LIN {X 0,Y 574.061,Z 827.419,A -85,B 0,C 180,E1 26876.471,E2 26876.471} C_VEL
LIN {X 0,Y 574.2,Z 764.795,A -85,B 0,C 180,E1 26875.555,E2 26875.555} C_VEL
LIN {X 0,Y 573.221,Z 758.441,A -85,B 0,C 180,E1 26875.376,E2 26875.376} C_VEL
LIN {X 0,Y 574.18,Z 705.798,A -85,B 0,C 180,E1 26872.197,E2 26872.197} C_VEL
LIN {X 0,Y 574.377,Z 695.779,A -85,B 0,C 180,E1 26871.578,E2 26871.578} C_VEL
LIN {X 0,Y 575.933,Z 695.849,A -85,B 0,C 180,E1 26871.383,E2 26871.383} C_VEL
LIN {X 0,Y 578.516,Z 693.344,A -85,B 0,C 180,E1 26871.064,E2 26871.064} C_VEL
LIN {X 0,Y 581.773,Z 687.657,A -85,B 0,C 180,E1 26870.669,E2 26870.669} C_VEL
LIN {X 0,Y 581.964,Z 745.865,A -85,B 0,C 180,E1 26870.646,E2 26870.646} C_VEL
LIN {X 0,Y 583.12,Z 759.023,A -85,B 0,C 180,E1 26870.508,E2 26870.508} C_VEL
LIN {X 0,Y 585.252,Z 769.853,A -85,B 0,C 180,E1 26870.255,E2 26870.255} C_VEL
LIN {X 0,Y 588.38,Z 779.136,A -85,B 0,C 180,E1 26869.89,E2 26869.89} C_VEL
LIN {X 0,Y 592.368,Z 786.864,A -85,B 0,C 180,E1 26869.429,E2 26869.429} C_VEL
LIN {X 0,Y 594.678,Z 791.282,A -85,B 0,C 180,E1 26868.994,E2 26868.994} C_VEL
LIN {X 0,Y 595.801,Z 794.66,A -85,B 0,C 180,E1 26868.457,E2 26868.457} C_VEL
LIN {X 0,Y 595.651,Z 796.735,A -85,B 0,C 180,E1 26867.897,E2 26867.897} C_VEL
LIN {X 0,Y 594.355,Z 797.607,A -85,B 0,C 180,E1 26867.317,E2 26867.317} C_VEL
LIN {X 0,Y 591.913,Z 797.089,A -85,B 0,C 180,E1 26866.722,E2 26866.722} C_VEL
LIN {X 0,Y 588.782,Z 795.144,A -85,B 0,C 180,E1 26866.197,E2 26866.197} C_VEL
LIN {X 0,Y 584.208,Z 790.552,A -85,B 0,C 180,E1 26865.535,E2 26865.535} C_VEL
LIN {X 0,Y 580.364,Z 783.96,A -85,B 0,C 180,E1 26864.799,E2 26864.799} C_VEL
LIN {X 0,Y 577.598,Z 774.842,A -85,B 0,C 180,E1 26863.96,E2 26863.96} C_VEL
LIN {X 0,Y 576.214,Z 763.514,A -85,B 0,C 180,E1 26863.07,E2 26863.07} C_VEL
LIN {X 0,Y 576.201,Z 743.269,A -85,B 0,C 180,E1 26861.695,E2 26861.695} C_VEL
LIN {X 0,Y 577.123,Z 706.105,A -85,B 0,C 180,E1 26859.16,E2 26859.16} C_VEL
LIN {X 0,Y 577.781,Z 682.335,A -85,B 0,C 180,E1 26857.465,E2 26857.465} C_VEL
LIN {X 0,Y 572.74,Z 672.999,A -85,B 0,C 180,E1 26856.161,E2 26856.161} C_VEL
LIN {X 0,Y 570.173,Z 668.299,A -85,B 0,C 180,E1 26855.481,E2 26855.481} C_VEL
LIN {X 0,Y 568.395,Z 664.903,A -85,B 0,C 180,E1 26854.992,E2 26854.992} C_VEL
LIN {X 0,Y 568.214,Z 663.961,A -85,B 0,C 180,E1 26854.882,E2 26854.882} C_VEL
LIN {X 0,Y 568.211,Z 663.959,A -85,B 0,C 180,E1 26851.607,E2 26851.607} C_VEL
LIN {X 0,Y 568.205,Z 663.957,A -85,B 0,C 180,E1 26848.252,E2 26848.252} C_VEL
LIN {X 0,Y 568.203,Z 663.955,A -85,B 0,C 180,E1 26844.981,E2 26844.981} C_VEL
LIN {X 0,Y 568.209,Z 663.955,A -85,B 0,C 180,E1 26841.686,E2 26841.686} C_VEL
LIN {X 0,Y 568.205,Z 663.957,A -85,B 0,C 180,E1 26838.466,E2 26838.466} C_VEL
LIN {X 0,Y 568.22,Z 663.957,A -85,B 0,C 180,E1 26835.2,E2 26835.2} C_VEL
LIN {X 0,Y 568.219,Z 663.959,A -85,B 0,C 180,E1 26831.881,E2 26831.881} C_VEL
LIN {X 0,Y 568.204,Z 663.958,A -85,B 0,C 180,E1 26828.602,E2 26828.602} C_VEL
LIN {X 0,Y 568.207,Z 663.956,A -85,B 0,C 180,E1 26825.351,E2 26825.351} C_VEL
LIN {X 0,Y 568.2,Z 663.956,A -85,B 0,C 180,E1 26822.118,E2 26822.118} C_VEL
LIN {X 0,Y 568.201,Z 663.956,A -85,B 0,C 180,E1 26818.891,E2 26818.891} C_VEL
LIN {X 0,Y 568.2,Z 663.956,A -85,B 0,C 180,E1 26815.66,E2 26815.66} C_VEL
LIN {X 0,Y 568.2,Z 663.957,A -85,B 0,C 180,E1 26812.416,E2 26812.416} C_VEL
LIN {X 0,Y 568.209,Z 663.957,A -85,B 0,C 180,E1 26809.147,E2 26809.147} C_VEL
LIN {X 0,Y 568.212,Z 663.958,A -85,B 0,C 180,E1 26805.842,E2 26805.842} C_VEL
LIN {X 0,Y 568.217,Z 663.957,A -85,B 0,C 180,E1 26802.488,E2 26802.488} C_VEL
LIN {X 0,Y 568.211,Z 663.955,A -85,B 0,C 180,E1 26799.815,E2 26799.815} C_VEL
LIN {X 0,Y 567.229,Z 664.083,A -85,B 0,C 180,E1 26799.039,E2 26799.039} C_VEL
LIN {X 0,Y 560.723,Z 664.89,A -85,B 0,C 180,E1 26796.802,E2 26796.802} C_VEL
LIN {X 0,Y 560.27,Z 664.947,A -85,B 0,C 180,E1 26796.29,E2 26796.29} C_VEL
LIN {X 0,Y 560.272,Z 664.94,A -85,B 0,C 180,E1 26793.045,E2 26793.045} C_VEL
LIN {X 0,Y 560.263,Z 664.941,A -85,B 0,C 180,E1 26789.74,E2 26789.74} C_VEL
LIN {X 0,Y 560.264,Z 664.943,A -85,B 0,C 180,E1 26786.45,E2 26786.45} C_VEL
LIN {X 0,Y 560.265,Z 664.941,A -85,B 0,C 180,E1 26783.156,E2 26783.156} C_VEL
LIN {X 0,Y 560.267,Z 664.943,A -85,B 0,C 180,E1 26779.891,E2 26779.891} C_VEL
LIN {X 0,Y 560.276,Z 664.948,A -85,B 0,C 180,E1 26776.578,E2 26776.578} C_VEL
LIN {X 0,Y 560.285,Z 664.95,A -85,B 0,C 180,E1 26773.256,E2 26773.256} C_VEL
LIN {X 0,Y 560.279,Z 664.95,A -85,B 0,C 180,E1 26769.84,E2 26769.84} C_VEL
LIN {X 0,Y 560.292,Z 665.024,A -85,B 0,C 180,E1 26767.165,E2 26767.165} C_VEL
LIN {X 0,Y 566.144,Z 680.018,A -85,B 0,C 180,E1 26765.71,E2 26765.71} C_VEL
LIN {X 0,Y 565.24,Z 725.275,A -85,B 0,C 180,E1 26762.648,E2 26762.648} C_VEL
LIN {X 0,Y 564.523,Z 766.047,A -85,B 0,C 180,E1 26759.972,E2 26759.972} C_VEL
LIN {X 0,Y 565.697,Z 774.516,A -85,B 0,C 180,E1 26759.782,E2 26759.782} C_VEL
LIN {X 0,Y 564.529,Z 1010.135,A -85,B 0,C 180,E1 26756.517,E2 26756.517} C_VEL
LIN {X 0,Y 564.318,Z 1034.29,A -85,B 0,C 180,E1 26756.118,E2 26756.118} C_VEL
LIN {X 0,Y 563.978,Z 1055.272,A -85,B 0,C 180,E1 26755.57,E2 26755.57} C_VEL
LIN {X 0,Y 563.594,Z 1074.97,A -85,B 0,C 180,E1 26754.863,E2 26754.863} C_VEL
LIN {X 0,Y 563.134,Z 1093.888,A -85,B 0,C 180,E1 26753.991,E2 26753.991} C_VEL
LIN {X 0,Y 562.646,Z 1111.983,A -85,B 0,C 180,E1 26752.964,E2 26752.964} C_VEL
LIN {X 0,Y 562.137,Z 1130.277,A -85,B 0,C 180,E1 26751.713,E2 26751.713} C_VEL
LIN {X 0,Y 561.654,Z 1147.441,A -85,B 0,C 180,E1 26750.312,E2 26750.312} C_VEL
LIN {X 0,Y 561.203,Z 1163.492,A -85,B 0,C 180,E1 26748.763,E2 26748.763} C_VEL
LIN {X 0,Y 560.824,Z 1178.065,A -85,B 0,C 180,E1 26747.107,E2 26747.107} C_VEL
LIN {X 0,Y 560.51,Z 1191.489,A -85,B 0,C 180,E1 26745.307,E2 26745.307} C_VEL
LIN {X 0,Y 560.275,Z 1203.372,A -85,B 0,C 180,E1 26743.414,E2 26743.414} C_VEL
LIN {X 0,Y 560.11,Z 1213.696,A -85,B 0,C 180,E1 26741.428,E2 26741.428} C_VEL
LIN {X 0,Y 560.004,Z 1222.013,A -85,B 0,C 180,E1 26739.454,E2 26739.454} C_VEL
LIN {X 0,Y 559.938,Z 1228.879,A -85,B 0,C 180,E1 26737.386,E2 26737.386} C_VEL
LIN {X 0,Y 559.914,Z 1234.17,A -85,B 0,C 180,E1 26735.225,E2 26735.225} C_VEL
LIN {X 0,Y 559.913,Z 1237.506,A -85,B 0,C 180,E1 26733.173,E2 26733.173} C_VEL
LIN {X 0,Y 559.912,Z 1239.241,A -85,B 0,C 180,E1 26731.125,E2 26731.125} C_VEL
LIN {X 0,Y 559.914,Z 1239.294,A -85,B 0,C 180,E1 26728.976,E2 26728.976} C_VEL
LIN {X 0,Y 559.914,Z 1237.717,A -85,B 0,C 180,E1 26726.929,E2 26726.929} C_VEL
LIN {X 0,Y 559.914,Z 1234.347,A -85,B 0,C 180,E1 26724.774,E2 26724.774} C_VEL
LIN {X 0,Y 559.934,Z 1229.439,A -85,B 0,C 180,E1 26722.716,E2 26722.716} C_VEL
LIN {X 0,Y 559.991,Z 1222.758,A -85,B 0,C 180,E1 26720.649,E2 26720.649} C_VEL
LIN {X 0,Y 560.099,Z 1214.577,A -85,B 0,C 180,E1 26718.675,E2 26718.675} C_VEL
LIN {X 0,Y 560.243,Z 1205.016,A -85,B 0,C 180,E1 26716.794,E2 26716.794} C_VEL
LIN {X 0,Y 560.463,Z 1193.494,A -85,B 0,C 180,E1 26714.902,E2 26714.902} C_VEL
LIN {X 0,Y 560.762,Z 1180.465,A -85,B 0,C 180,E1 26713.104,E2 26713.104} C_VEL
LIN {X 0,Y 561.151,Z 1165.383,A -85,B 0,C 180,E1 26711.347,E2 26711.347} C_VEL
LIN {X 0,Y 561.596,Z 1149.282,A -85,B 0,C 180,E1 26709.763,E2 26709.763} C_VEL
LIN {X 0,Y 562.058,Z 1132.894,A -85,B 0,C 180,E1 26708.393,E2 26708.393} C_VEL
LIN {X 0,Y 562.578,Z 1115.255,A -85,B 0,C 180,E1 26707.149,E2 26707.149} C_VEL
LIN {X 0,Y 563.08,Z 1096.267,A -85,B 0,C 180,E1 26706.042,E2 26706.042} C_VEL
LIN {X 0,Y 563.532,Z 1076.995,A -85,B 0,C 180,E1 26705.133,E2 26705.133} C_VEL
LIN {X 0,Y 563.952,Z 1056.45,A -85,B 0,C 180,E1 26704.378,E2 26704.378} C_VEL
LIN {X 0,Y 564.303,Z 1035.559,A -85,B 0,C 180,E1 26703.82,E2 26703.82} C_VEL
LIN {X 0,Y 564.518,Z 1012.48,A -85,B 0,C 180,E1 26703.425,E2 26703.425} C_VEL
LIN {X 0,Y 565.69,Z 776.957,A -85,B 0,C 180,E1 26700.162,E2 26700.162} C_VEL
LIN {X 0,Y 563.542,Z 767.47,A -85,B 0,C 180,E1 26699.888,E2 26699.888} C_VEL
LIN {X 0,Y 564.325,Z 733.661,A -85,B 0,C 180,E1 26696.684,E2 26696.684} C_VEL
LIN {X 0,Y 565.011,Z 702.166,A -85,B 0,C 180,E1 26693.628,E2 26693.628} C_VEL
LIN {X 0,Y 565.36,Z 679.55,A -85,B 0,C 180,E1 26691.416,E2 26691.416} C_VEL
LIN {X 0,Y 560.271,Z 664.95,A -85,B 0,C 180,E1 26689.556,E2 26689.556} C_VEL
LIN {X 0,Y 560.272,Z 664.947,A -85,B 0,C 180,E1 26686.178,E2 26686.178} C_VEL
LIN {X 0,Y 560.267,Z 664.94,A -85,B 0,C 180,E1 26682.821,E2 26682.821} C_VEL
LIN {X 0,Y 560.281,Z 664.944,A -85,B 0,C 180,E1 26679.401,E2 26679.401} C_VEL
LIN {X 0,Y 560.283,Z 664.949,A -85,B 0,C 180,E1 26675.953,E2 26675.953} C_VEL
LIN {X 0,Y 560.289,Z 665.066,A -85,B 0,C 180,E1 26674.08,E2 26674.08} C_VEL
LIN {X 0,Y 565.192,Z 678.885,A -85,B 0,C 180,E1 26672.474,E2 26672.474} C_VEL
LIN {X 0,Y 563.991,Z 718.046,A -85,B 0,C 180,E1 26669.12,E2 26669.12} C_VEL
LIN {X 0,Y 563.138,Z 756.776,A -85,B 0,C 180,E1 26665.955,E2 26665.955} C_VEL
LIN {X 0,Y 562.433,Z 797.021,A -85,B 0,C 180,E1 26662.762,E2 26662.762} C_VEL
LIN {X 0,Y 561.797,Z 839.094,A -85,B 0,C 180,E1 26659.494,E2 26659.494} C_VEL
LIN {X 0,Y 561.794,Z 845.338,A -85,B 0,C 180,E1 26659.043,E2 26659.043} C_VEL
LIN {X 0,Y 562.522,Z 852.682,A -85,B 0,C 180,E1 26658.919,E2 26658.919} C_VEL
LIN {X 0,Y 561.965,Z 1014.791,A -85,B 0,C 180,E1 26656.766,E2 26656.766} C_VEL
LIN {X 0,Y 561.803,Z 1032.643,A -85,B 0,C 180,E1 26656.339,E2 26656.339} C_VEL
LIN {X 0,Y 561.572,Z 1048.909,A -85,B 0,C 180,E1 26655.755,E2 26655.755} C_VEL
LIN {X 0,Y 561.319,Z 1064.386,A -85,B 0,C 180,E1 26655.021,E2 26655.021} C_VEL
LIN {X 0,Y 561.035,Z 1079.974,A -85,B 0,C 180,E1 26654.08,E2 26654.08} C_VEL
LIN {X 0,Y 560.761,Z 1094.334,A -85,B 0,C 180,E1 26652.983,E2 26652.983} C_VEL
LIN {X 0,Y 560.523,Z 1107.266,A -85,B 0,C 180,E1 26651.786,E2 26651.786} C_VEL
LIN {X 0,Y 560.306,Z 1119.603,A -85,B 0,C 180,E1 26650.384,E2 26650.384} C_VEL
LIN {X 0,Y 560.145,Z 1129.955,A -85,B 0,C 180,E1 26648.934,E2 26648.934} C_VEL
LIN {X 0,Y 560.038,Z 1138.965,A -85,B 0,C 180,E1 26647.386,E2 26647.386} C_VEL
LIN {X 0,Y 559.961,Z 1146.839,A -85,B 0,C 180,E1 26645.636,E2 26645.636} C_VEL
LIN {X 0,Y 559.93,Z 1152.371,A -85,B 0,C 180,E1 26643.994,E2 26643.994} C_VEL
LIN {X 0,Y 559.915,Z 1156.495,A -85,B 0,C 180,E1 26642.252,E2 26642.252} C_VEL
LIN {X 0,Y 559.916,Z 1158.797,A -85,B 0,C 180,E1 26640.512,E2 26640.512} C_VEL
LIN {X 0,Y 559.913,Z 1159.457,A -85,B 0,C 180,E1 26638.772,E2 26638.772} C_VEL
LIN {X 0,Y 559.913,Z 1158.352,A -85,B 0,C 180,E1 26636.929,E2 26636.929} C_VEL
LIN {X 0,Y 559.921,Z 1155.476,A -85,B 0,C 180,E1 26635.158,E2 26635.158} C_VEL
LIN {X 0,Y 559.934,Z 1151.257,A -85,B 0,C 180,E1 26633.541,E2 26633.541} C_VEL
LIN {X 0,Y 559.975,Z 1145.334,A -85,B 0,C 180,E1 26631.891,E2 26631.891} C_VEL
LIN {X 0,Y 560.047,Z 1137.357,A -85,B 0,C 180,E1 26630.229,E2 26630.229} C_VEL
LIN {X 0,Y 560.163,Z 1128.687,A -85,B 0,C 180,E1 26628.781,E2 26628.781} C_VEL
LIN {X 0,Y 560.348,Z 1117.102,A -85,B 0,C 180,E1 26627.217,E2 26627.217} C_VEL
LIN {X 0,Y 560.556,Z 1105.086,A -85,B 0,C 180,E1 26625.909,E2 26625.909} C_VEL
LIN {X 0,Y 560.804,Z 1092.283,A -85,B 0,C 180,E1 26624.753,E2 26624.753} C_VEL
LIN {X 0,Y 561.11,Z 1076.384,A -85,B 0,C 180,E1 26623.595,E2 26623.595} C_VEL
LIN {X 0,Y 561.365,Z 1061.702,A -85,B 0,C 180,E1 26622.749,E2 26622.749} C_VEL
LIN {X 0,Y 561.612,Z 1046.666,A -85,B 0,C 180,E1 26622.062,E2 26622.062} C_VEL
LIN {X 0,Y 561.851,Z 1028.62,A -85,B 0,C 180,E1 26621.459,E2 26621.459} C_VEL
LIN {X 0,Y 561.993,Z 1012.392,A -85,B 0,C 180,E1 26621.104,E2 26621.104} C_VEL
LIN {X 0,Y 562.344,Z 849.073,A -85,B 0,C 180,E1 26618.937,E2 26618.937} C_VEL
LIN {X 0,Y 561.734,Z 844.641,A -85,B 0,C 180,E1 26618.843,E2 26618.843} C_VEL
LIN {X 0,Y 562.377,Z 801.196,A -85,B 0,C 180,E1 26615.476,E2 26615.476} C_VEL
LIN {X 0,Y 563.114,Z 758.703,A -85,B 0,C 180,E1 26612.11,E2 26612.11} C_VEL
LIN {X 0,Y 563.618,Z 737.518,A -85,B 0,C 180,E1 26610.373,E2 26610.373} C_VEL
LIN {X 0,Y 566.841,Z 712.359,A -85,B 0,C 180,E1 26607.812,E2 26607.812} C_VEL
LIN {X 0,Y 571.277,Z 691.502,A -85,B 0,C 180,E1 26605.523,E2 26605.523} C_VEL
LIN {X 0,Y 572.681,Z 686.32,A -85,B 0,C 180,E1 26604.881,E2 26604.881} C_VEL
LIN {X 0,Y 571.086,Z 683.566,A -85,B 0,C 180,E1 26603.343,E2 26603.343} C_VEL
LIN {X 0,Y 571.107,Z 682.763,A -85,B 0,C 180,E1 26602.338,E2 26602.338} C_VEL
LIN {X 0,Y 571.316,Z 684.023,A -85,B 0,C 180,E1 26601.526,E2 26601.526} C_VEL
LIN {X 0,Y 571.112,Z 684.711,A -85,B 0,C 180,E1 26601.425,E2 26601.425} C_VEL
LIN {X 0,Y 567.688,Z 695.309,A -85,B 0,C 180,E1 26600.563,E2 26600.563} C_VEL
LIN {X 0,Y 565.443,Z 708.541,A -85,B 0,C 180,E1 26599.652,E2 26599.652} C_VEL
LIN {X 0,Y 563.893,Z 729.692,A -85,B 0,C 180,E1 26598.398,E2 26598.398} C_VEL
LIN {X 0,Y 564.008,Z 751.659,A -85,B 0,C 180,E1 26597.175,E2 26597.175} C_VEL
LIN {X 0,Y 565.908,Z 767.995,A -85,B 0,C 180,E1 26596.235,E2 26596.235} C_VEL
LIN {X 0,Y 569.138,Z 779.936,A -85,B 0,C 180,E1 26595.496,E2 26595.496} C_VEL
LIN {X 0,Y 573.479,Z 789.298,A -85,B 0,C 180,E1 26594.869,E2 26594.869} C_VEL
LIN {X 0,Y 578.552,Z 796.38,A -85,B 0,C 180,E1 26594.318,E2 26594.318} C_VEL
LIN {X 0,Y 582.873,Z 800.653,A -85,B 0,C 180,E1 26593.907,E2 26593.907} C_VEL
LIN {X 0,Y 586.666,Z 803.361,A -85,B 0,C 180,E1 26593.445,E2 26593.445} C_VEL
LIN {X 0,Y 589.834,Z 804.737,A -85,B 0,C 180,E1 26592.92,E2 26592.92} C_VEL
LIN {X 0,Y 592.243,Z 804.795,A -85,B 0,C 180,E1 26592.315,E2 26592.315} C_VEL
LIN {X 0,Y 593.403,Z 803.535,A -85,B 0,C 180,E1 26591.718,E2 26591.718} C_VEL
LIN {X 0,Y 593.289,Z 801.151,A -85,B 0,C 180,E1 26591.149,E2 26591.149} C_VEL
LIN {X 0,Y 591.814,Z 797.58,A -85,B 0,C 180,E1 26590.617,E2 26590.617} C_VEL
LIN {X 0,Y 589.03,Z 792.986,A -85,B 0,C 180,E1 26590.185,E2 26590.185} C_VEL
LIN {X 0,Y 584.618,Z 784.743,A -85,B 0,C 180,E1 26589.67,E2 26589.67} C_VEL
LIN {X 0,Y 581.163,Z 775.111,A -85,B 0,C 180,E1 26589.257,E2 26589.257} C_VEL
LIN {X 0,Y 578.719,Z 764.246,A -85,B 0,C 180,E1 26588.96,E2 26588.96} C_VEL
LIN {X 0,Y 577.209,Z 751.284,A -85,B 0,C 180,E1 26588.775,E2 26588.775} C_VEL
LIN {X 0,Y 576.744,Z 738.293,A -85,B 0,C 180,E1 26588.717,E2 26588.717} C_VEL
LIN {X 0,Y 576.681,Z 705.582,A -85,B 0,C 180,E1 26588.709,E2 26588.709} C_VEL
LIN {X 0,Y 572.755,Z 714.129,A -85,B 0,C 180,E1 26588.217,E2 26588.217} C_VEL
LIN {X 0,Y 569.752,Z 718.329,A -85,B 0,C 180,E1 26587.832,E2 26587.832} C_VEL
LIN {X 0,Y 568.223,Z 719.281,A -85,B 0,C 180,E1 26587.632,E2 26587.632} C_VEL
LIN {X 0,Y 567.239,Z 719.066,A -85,B 0,C 180,E1 26587.502,E2 26587.502} C_VEL
LIN {X 0,Y 566.472,Z 759.406,A -85,B 0,C 180,E1 26585.065,E2 26585.065} C_VEL
LIN {X 0,Y 567.771,Z 768.747,A -85,B 0,C 180,E1 26584.832,E2 26584.832} C_VEL
LIN {X 0,Y 566.351,Z 1004.078,A -85,B 0,C 180,E1 26581.438,E2 26581.438} C_VEL
LIN {X 0,Y 565.933,Z 1066.266,A -85,B 0,C 180,E1 26580.527,E2 26580.527} C_VEL
LIN {X 0,Y 565.555,Z 1088.579,A -85,B 0,C 180,E1 26580.002,E2 26580.002} C_VEL
LIN {X 0,Y 565.047,Z 1110.998,A -85,B 0,C 180,E1 26579.265,E2 26579.265} C_VEL
LIN {X 0,Y 564.539,Z 1131.562,A -85,B 0,C 180,E1 26578.395,E2 26578.395} C_VEL
LIN {X 0,Y 563.916,Z 1151.757,A -85,B 0,C 180,E1 26577.337,E2 26577.337} C_VEL
LIN {X 0,Y 563.287,Z 1171.672,A -85,B 0,C 180,E1 26576.082,E2 26576.082} C_VEL
LIN {X 0,Y 562.667,Z 1190.469,A -85,B 0,C 180,E1 26574.683,E2 26574.683} C_VEL
LIN {X 0,Y 562.059,Z 1208.4,A -85,B 0,C 180,E1 26573.118,E2 26573.118} C_VEL
LIN {X 0,Y 561.559,Z 1224.188,A -85,B 0,C 180,E1 26571.518,E2 26571.518} C_VEL
LIN {X 0,Y 561.086,Z 1239.886,A -85,B 0,C 180,E1 26569.682,E2 26569.682} C_VEL
LIN {X 0,Y 560.71,Z 1254.044,A -85,B 0,C 180,E1 26567.754,E2 26567.754} C_VEL
LIN {X 0,Y 560.408,Z 1266.743,A -85,B 0,C 180,E1 26565.736,E2 26565.736} C_VEL
LIN {X 0,Y 560.192,Z 1277.859,A -85,B 0,C 180,E1 26563.627,E2 26563.627} C_VEL
LIN {X 0,Y 560.053,Z 1287.491,A -85,B 0,C 180,E1 26561.43,E2 26561.43} C_VEL
LIN {X 0,Y 559.975,Z 1295.228,A -85,B 0,C 180,E1 26559.248,E2 26559.248} C_VEL
LIN {X 0,Y 559.928,Z 1300.904,A -85,B 0,C 180,E1 26557.181,E2 26557.181} C_VEL
LIN {X 0,Y 559.906,Z 1305.479,A -85,B 0,C 180,E1 26554.918,E2 26554.918} C_VEL
LIN {X 0,Y 559.9,Z 1308.314,A -85,B 0,C 180,E1 26552.662,E2 26552.662} C_VEL
LIN {X 0,Y 559.894,Z 1309.395,A -85,B 0,C 180,E1 26550.512,E2 26550.512} C_VEL
LIN {X 0,Y 559.899,Z 1308.894,A -85,B 0,C 180,E1 26548.158,E2 26548.158} C_VEL
LIN {X 0,Y 559.9,Z 1306.853,A -85,B 0,C 180,E1 26546.007,E2 26546.007} C_VEL
LIN {X 0,Y 559.908,Z 1303.407,A -85,B 0,C 180,E1 26543.953,E2 26543.953} C_VEL
LIN {X 0,Y 559.942,Z 1297.983,A -85,B 0,C 180,E1 26541.684,E2 26541.684} C_VEL
LIN {X 0,Y 560.003,Z 1291.416,A -85,B 0,C 180,E1 26539.612,E2 26539.612} C_VEL
LIN {X 0,Y 560.111,Z 1282.696,A -85,B 0,C 180,E1 26537.422,E2 26537.422} C_VEL
LIN {X 0,Y 560.286,Z 1272.365,A -85,B 0,C 180,E1 26535.289,E2 26535.289} C_VEL
LIN {X 0,Y 560.529,Z 1261.619,A -85,B 0,C 180,E1 26533.418,E2 26533.418} C_VEL
LIN {X 0,Y 560.865,Z 1248.037,A -85,B 0,C 180,E1 26531.392,E2 26531.392} C_VEL
LIN {X 0,Y 561.288,Z 1232.807,A -85,B 0,C 180,E1 26529.456,E2 26529.456} C_VEL
LIN {X 0,Y 561.785,Z 1217.032,A -85,B 0,C 180,E1 26527.723,E2 26527.723} C_VEL
LIN {X 0,Y 562.372,Z 1199.159,A -85,B 0,C 180,E1 26526.043,E2 26526.043} C_VEL
LIN {X 0,Y 562.97,Z 1181.221,A -85,B 0,C 180,E1 26524.602,E2 26524.602} C_VEL
LIN {X 0,Y 563.597,Z 1161.906,A -85,B 0,C 180,E1 26523.275,E2 26523.275} C_VEL
LIN {X 0,Y 564.221,Z 1141.648,A -85,B 0,C 180,E1 26522.107,E2 26522.107} C_VEL
LIN {X 0,Y 564.832,Z 1120.938,A -85,B 0,C 180,E1 26521.131,E2 26521.131} C_VEL
LIN {X 0,Y 565.313,Z 1099.125,A -85,B 0,C 180,E1 26520.319,E2 26520.319} C_VEL
LIN {X 0,Y 565.78,Z 1076.989,A -85,B 0,C 180,E1 26519.7,E2 26519.7} C_VEL
LIN {X 0,Y 566.051,Z 1054.545,A -85,B 0,C 180,E1 26519.277,E2 26519.277} C_VEL
LIN {X 0,Y 567.388,Z 827.927,A -85,B 0,C 180,E1 26516.031,E2 26516.031} C_VEL
LIN {X 0,Y 567.58,Z 766.128,A -85,B 0,C 180,E1 26515.115,E2 26515.115} C_VEL
LIN {X 0,Y 566.384,Z 758.441,A -85,B 0,C 180,E1 26514.897,E2 26514.897} C_VEL
LIN {X 0,Y 567.303,Z 719.089,A -85,B 0,C 180,E1 26512.488,E2 26512.488} C_VEL
LIN {X 0,Y 568.829,Z 719.046,A -85,B 0,C 180,E1 26512.289,E2 26512.289} C_VEL
LIN {X 0,Y 571.437,Z 716.257,A -85,B 0,C 180,E1 26511.951,E2 26511.951} C_VEL
LIN {X 0,Y 575.154,Z 709.281,A -85,B 0,C 180,E1 26511.481,E2 26511.481} C_VEL
LIN {X 0,Y 576.739,Z 705.432,A -85,B 0,C 180,E1 26511.283,E2 26511.283} C_VEL
LIN {X 0,Y 576.939,Z 746.497,A -85,B 0,C 180,E1 26511.259,E2 26511.259} C_VEL
LIN {X 0,Y 578.105,Z 760.159,A -85,B 0,C 180,E1 26511.115,E2 26511.115} C_VEL
LIN {X 0,Y 580.288,Z 771.863,A -85,B 0,C 180,E1 26510.848,E2 26510.848} C_VEL
LIN {X 0,Y 583.457,Z 781.953,A -85,B 0,C 180,E1 26510.468,E2 26510.468} C_VEL
LIN {X 0,Y 587.575,Z 790.606,A -85,B 0,C 180,E1 26509.984,E2 26509.984} C_VEL
LIN {X 0,Y 591.165,Z 796.381,A -85,B 0,C 180,E1 26509.515,E2 26509.515} C_VEL
LIN {X 0,Y 593,Z 800.231,A -85,B 0,C 180,E1 26509.013,E2 26509.013} C_VEL
LIN {X 0,Y 593.488,Z 803.086,A -85,B 0,C 180,E1 26508.418,E2 26508.418} C_VEL
LIN {X 0,Y 592.548,Z 804.664,A -85,B 0,C 180,E1 26507.796,E2 26507.796} C_VEL
LIN {X 0,Y 590.294,Z 804.841,A -85,B 0,C 180,E1 26507.174,E2 26507.174} C_VEL
LIN {X 0,Y 587.239,Z 803.679,A -85,B 0,C 180,E1 26506.637,E2 26506.637} C_VEL
LIN {X 0,Y 582.393,Z 800.238,A -85,B 0,C 180,E1 26506,E2 26506} C_VEL
LIN {X 0,Y 577.407,Z 794.531,A -85,B 0,C 180,E1 26505.232,E2 26505.232} C_VEL
LIN {X 0,Y 573.569,Z 786.965,A -85,B 0,C 180,E1 26504.419,E2 26504.419} C_VEL
LIN {X 0,Y 570.992,Z 777.221,A -85,B 0,C 180,E1 26503.536,E2 26503.536} C_VEL
LIN {X 0,Y 569.797,Z 765.733,A -85,B 0,C 180,E1 26502.636,E2 26502.636} C_VEL
LIN {X 0,Y 570.054,Z 741.784,A -85,B 0,C 180,E1 26500.994,E2 26500.994} C_VEL
LIN {X 0,Y 571.13,Z 706.577,A -85,B 0,C 180,E1 26498.553,E2 26498.553} C_VEL
LIN {X 0,Y 571.671,Z 686.823,A -85,B 0,C 180,E1 26497.114,E2 26497.114} C_VEL
LIN {X 0,Y 565.079,Z 674.321,A -85,B 0,C 180,E1 26495.345,E2 26495.345} C_VEL
LIN {X 0,Y 562.956,Z 670.34,A -85,B 0,C 180,E1 26494.759,E2 26494.759} C_VEL
LIN {X 0,Y 560.669,Z 666.627,A -85,B 0,C 180,E1 26494.162,E2 26494.162} C_VEL
LIN {X 0,Y 560.28,Z 664.949,A -85,B 0,C 180,E1 26493.957,E2 26493.957} C_VEL
LIN {X 0,Y 560.287,Z 664.946,A -85,B 0,C 180,E1 26490.57,E2 26490.57} C_VEL
LIN {X 0,Y 560.274,Z 664.941,A -85,B 0,C 180,E1 26487.184,E2 26487.184} C_VEL
LIN {X 0,Y 560.265,Z 664.945,A -85,B 0,C 180,E1 26483.898,E2 26483.898} C_VEL
LIN {X 0,Y 560.266,Z 664.945,A -85,B 0,C 180,E1 26480.692,E2 26480.692} C_VEL
LIN {X 0,Y 560.265,Z 664.944,A -85,B 0,C 180,E1 26477.446,E2 26477.446} C_VEL
LIN {X 0,Y 560.264,Z 664.945,A -85,B 0,C 180,E1 26474.152,E2 26474.152} C_VEL
LIN {X 0,Y 560.27,Z 664.946,A -85,B 0,C 180,E1 26470.8,E2 26470.8} C_VEL
LIN {X 0,Y 560.268,Z 664.948,A -85,B 0,C 180,E1 26467.485,E2 26467.485} C_VEL
LIN {X 0,Y 560.279,Z 664.947,A -85,B 0,C 180,E1 26464.196,E2 26464.196} C_VEL
LIN {X 0,Y 560.279,Z 664.944,A -85,B 0,C 180,E1 26460.818,E2 26460.818} C_VEL
LIN {X 0,Y 560.273,Z 664.944,A -85,B 0,C 180,E1 26457.443,E2 26457.443} C_VEL
LIN {X 0,Y 560.281,Z 664.943,A -85,B 0,C 180,E1 26453.956,E2 26453.956} C_VEL
LIN {X 0,Y 560.275,Z 664.946,A -85,B 0,C 180,E1 26450.55,E2 26450.55} C_VEL
LIN {X 0,Y 560.277,Z 664.947,A -85,B 0,C 180,E1 26447.215,E2 26447.215} C_VEL
LIN {X 0,Y 560.273,Z 664.946,A -85,B 0,C 180,E1 26443.942,E2 26443.942} C_VEL
LIN {X 0,Y 560.263,Z 664.943,A -85,B 0,C 180,E1 26440.613,E2 26440.613} C_VEL
LIN {X 0,Y 560.261,Z 664.943,A -85,B 0,C 180,E1 26437.437,E2 26437.437} C_VEL
LIN {X 0,Y 560.27,Z 664.947,A -85,B 0,C 180,E1 26436.29,E2 26436.29} C_VEL
LIN {X 0,Y 559.258,Z 665.074,A -85,B 0,C 180,E1 26435.503,E2 26435.503} C_VEL
LIN {X 0,Y 552.854,Z 665.867,A -85,B 0,C 180,E1 26433.291,E2 26433.291} C_VEL
LIN {X 0,Y 552.337,Z 665.926,A -85,B 0,C 180,E1 26432.715,E2 26432.715} C_VEL
LIN {X 0,Y 552.344,Z 665.927,A -85,B 0,C 180,E1 26429.298,E2 26429.298} C_VEL
LIN {X 0,Y 552.346,Z 665.927,A -85,B 0,C 180,E1 26425.817,E2 26425.817} C_VEL
LIN {X 0,Y 552.338,Z 665.937,A -85,B 0,C 180,E1 26422.407,E2 26422.407} C_VEL
LIN {X 0,Y 552.324,Z 665.925,A -85,B 0,C 180,E1 26419.056,E2 26419.056} C_VEL
LIN {X 0,Y 552.324,Z 665.936,A -85,B 0,C 180,E1 26415.796,E2 26415.796} C_VEL
LIN {X 0,Y 552.324,Z 665.938,A -85,B 0,C 180,E1 26412.542,E2 26412.542} C_VEL
LIN {X 0,Y 552.324,Z 665.94,A -85,B 0,C 180,E1 26409.315,E2 26409.315} C_VEL
LIN {X 0,Y 552.349,Z 666.006,A -85,B 0,C 180,E1 26407.69,E2 26407.69} C_VEL
LIN {X 0,Y 559.187,Z 683.251,A -85,B 0,C 180,E1 26405.977,E2 26405.977} C_VEL
LIN {X 0,Y 558.193,Z 727.012,A -85,B 0,C 180,E1 26402.992,E2 26402.992} C_VEL
LIN {X 0,Y 557.384,Z 766.146,A -85,B 0,C 180,E1 26400.396,E2 26400.396} C_VEL
LIN {X 0,Y 558.749,Z 775.709,A -85,B 0,C 180,E1 26400.174,E2 26400.174} C_VEL
LIN {X 0,Y 557.367,Z 1011.261,A -85,B 0,C 180,E1 26396.87,E2 26396.87} C_VEL
LIN {X 0,Y 557.117,Z 1034.783,A -85,B 0,C 180,E1 26396.471,E2 26396.471} C_VEL
LIN {X 0,Y 556.725,Z 1055.687,A -85,B 0,C 180,E1 26395.915,E2 26395.915} C_VEL
LIN {X 0,Y 556.283,Z 1074.993,A -85,B 0,C 180,E1 26395.212,E2 26395.212} C_VEL
LIN {X 0,Y 555.713,Z 1094.996,A -85,B 0,C 180,E1 26394.275,E2 26394.275} C_VEL
LIN {X 0,Y 555.112,Z 1113.841,A -85,B 0,C 180,E1 26393.175,E2 26393.175} C_VEL
LIN {X 0,Y 554.518,Z 1131.728,A -85,B 0,C 180,E1 26391.915,E2 26391.915} C_VEL
LIN {X 0,Y 553.947,Z 1148.811,A -85,B 0,C 180,E1 26390.482,E2 26390.482} C_VEL
LIN {X 0,Y 553.407,Z 1165.059,A -85,B 0,C 180,E1 26388.868,E2 26388.868} C_VEL
LIN {X 0,Y 552.957,Z 1179.771,A -85,B 0,C 180,E1 26387.141,E2 26387.141} C_VEL
LIN {X 0,Y 552.592,Z 1192.908,A -85,B 0,C 180,E1 26385.317,E2 26385.317} C_VEL
LIN {X 0,Y 552.324,Z 1204.533,A -85,B 0,C 180,E1 26383.398,E2 26383.398} C_VEL
LIN {X 0,Y 552.142,Z 1214.188,A -85,B 0,C 180,E1 26381.489,E2 26381.489} C_VEL
LIN {X 0,Y 552.02,Z 1222.416,A -85,B 0,C 180,E1 26379.487,E2 26379.487} C_VEL
LIN {X 0,Y 551.951,Z 1228.882,A -85,B 0,C 180,E1 26377.494,E2 26377.494} C_VEL
LIN {X 0,Y 551.918,Z 1234.171,A -85,B 0,C 180,E1 26375.301,E2 26375.301} C_VEL
LIN {X 0,Y 551.913,Z 1237.507,A -85,B 0,C 180,E1 26373.219,E2 26373.219} C_VEL
LIN {X 0,Y 551.911,Z 1239.241,A -85,B 0,C 180,E1 26371.141,E2 26371.141} C_VEL
LIN {X 0,Y 551.914,Z 1239.293,A -85,B 0,C 180,E1 26368.962,E2 26368.962} C_VEL
LIN {X 0,Y 551.915,Z 1237.717,A -85,B 0,C 180,E1 26366.884,E2 26366.884} C_VEL
LIN {X 0,Y 551.917,Z 1234.346,A -85,B 0,C 180,E1 26364.698,E2 26364.698} C_VEL
LIN {X 0,Y 551.942,Z 1229.436,A -85,B 0,C 180,E1 26362.61,E2 26362.61} C_VEL
LIN {X 0,Y 552.012,Z 1222.754,A -85,B 0,C 180,E1 26360.512,E2 26360.512} C_VEL
LIN {X 0,Y 552.142,Z 1214.235,A -85,B 0,C 180,E1 26358.431,E2 26358.431} C_VEL
LIN {X 0,Y 552.332,Z 1203.86,A -85,B 0,C 180,E1 26356.388,E2 26356.388} C_VEL
LIN {X 0,Y 552.617,Z 1192.08,A -85,B 0,C 180,E1 26354.467,E2 26354.467} C_VEL
LIN {X 0,Y 552.985,Z 1178.77,A -85,B 0,C 180,E1 26352.642,E2 26352.642} C_VEL
LIN {X 0,Y 553.447,Z 1163.867,A -85,B 0,C 180,E1 26350.913,E2 26350.913} C_VEL
LIN {X 0,Y 553.978,Z 1147.819,A -85,B 0,C 180,E1 26349.338,E2 26349.338} C_VEL
LIN {X 0,Y 554.581,Z 1129.994,A -85,B 0,C 180,E1 26347.864,E2 26347.864} C_VEL
LIN {X 0,Y 555.169,Z 1112.038,A -85,B 0,C 180,E1 26346.622,E2 26346.622} C_VEL
LIN {X 0,Y 555.75,Z 1093.402,A -85,B 0,C 180,E1 26345.555,E2 26345.555} C_VEL
LIN {X 0,Y 556.312,Z 1073.883,A -85,B 0,C 180,E1 26344.652,E2 26344.652} C_VEL
LIN {X 0,Y 556.794,Z 1053.202,A -85,B 0,C 180,E1 26343.916,E2 26343.916} C_VEL
LIN {X 0,Y 557.146,Z 1032.357,A -85,B 0,C 180,E1 26343.386,E2 26343.386} C_VEL
LIN {X 0,Y 557.398,Z 1005.712,A -85,B 0,C 180,E1 26342.963,E2 26342.963} C_VEL
LIN {X 0,Y 558.721,Z 778.33,A -85,B 0,C 180,E1 26339.772,E2 26339.772} C_VEL
LIN {X 0,Y 556.242,Z 767.449,A -85,B 0,C 180,E1 26339.449,E2 26339.449} C_VEL
LIN {X 0,Y 557.206,Z 733.595,A -85,B 0,C 180,E1 26336.183,E2 26336.183} C_VEL
LIN {X 0,Y 557.942,Z 701.614,A -85,B 0,C 180,E1 26333.059,E2 26333.059} C_VEL
LIN {X 0,Y 558.173,Z 682.619,A -85,B 0,C 180,E1 26331.174,E2 26331.174} C_VEL
LIN {X 0,Y 552.345,Z 665.934,A -85,B 0,C 180,E1 26329.013,E2 26329.013} C_VEL
LIN {X 0,Y 552.337,Z 665.935,A -85,B 0,C 180,E1 26325.647,E2 26325.647} C_VEL
LIN {X 0,Y 552.341,Z 665.932,A -85,B 0,C 180,E1 26322.236,E2 26322.236} C_VEL
LIN {X 0,Y 552.326,Z 665.933,A -85,B 0,C 180,E1 26318.884,E2 26318.884} C_VEL
LIN {X 0,Y 552.328,Z 665.94,A -85,B 0,C 180,E1 26315.628,E2 26315.628} C_VEL
LIN {X 0,Y 552.328,Z 665.937,A -85,B 0,C 180,E1 26314.641,E2 26314.641} C_VEL
LIN {X 0,Y 558.19,Z 681.707,A -85,B 0,C 180,E1 26312.749,E2 26312.749} C_VEL
LIN {X 0,Y 556.876,Z 720.273,A -85,B 0,C 180,E1 26309.417,E2 26309.417} C_VEL
LIN {X 0,Y 555.692,Z 759.496,A -85,B 0,C 180,E1 26306.123,E2 26306.123} C_VEL
LIN {X 0,Y 554.853,Z 800.214,A -85,B 0,C 180,E1 26302.851,E2 26302.851} C_VEL
LIN {X 0,Y 554.095,Z 842.794,A -85,B 0,C 180,E1 26299.502,E2 26299.502} C_VEL
LIN {X 0,Y 554.148,Z 845.441,A -85,B 0,C 180,E1 26299.331,E2 26299.331} C_VEL
LIN {X 0,Y 555.001,Z 853.358,A -85,B 0,C 180,E1 26299.192,E2 26299.192} C_VEL
LIN {X 0,Y 554.348,Z 1014.486,A -85,B 0,C 180,E1 26297.023,E2 26297.023} C_VEL
LIN {X 0,Y 554.167,Z 1031.972,A -85,B 0,C 180,E1 26296.607,E2 26296.607} C_VEL
LIN {X 0,Y 553.904,Z 1048.016,A -85,B 0,C 180,E1 26296.033,E2 26296.033} C_VEL
LIN {X 0,Y 553.614,Z 1062.964,A -85,B 0,C 180,E1 26295.326,E2 26295.326} C_VEL
LIN {X 0,Y 553.281,Z 1078.623,A -85,B 0,C 180,E1 26294.389,E2 26294.389} C_VEL
LIN {X 0,Y 552.949,Z 1093.271,A -85,B 0,C 180,E1 26293.276,E2 26293.276} C_VEL
LIN {X 0,Y 552.669,Z 1105.841,A -85,B 0,C 180,E1 26292.114,E2 26292.114} C_VEL
LIN {X 0,Y 552.419,Z 1118.059,A -85,B 0,C 180,E1 26290.745,E2 26290.745} C_VEL
LIN {X 0,Y 552.213,Z 1128.698,A -85,B 0,C 180,E1 26289.274,E2 26289.274} C_VEL
LIN {X 0,Y 552.078,Z 1137.357,A -85,B 0,C 180,E1 26287.807,E2 26287.807} C_VEL
LIN {X 0,Y 551.991,Z 1145.28,A -85,B 0,C 180,E1 26286.135,E2 26286.135} C_VEL
LIN {X 0,Y 551.938,Z 1151.192,A -85,B 0,C 180,E1 26284.468,E2 26284.468} C_VEL
LIN {X 0,Y 551.919,Z 1155.476,A -85,B 0,C 180,E1 26282.804,E2 26282.804} C_VEL
LIN {X 0,Y 551.913,Z 1158.324,A -85,B 0,C 180,E1 26281.038,E2 26281.038} C_VEL
LIN {X 0,Y 551.914,Z 1159.45,A -85,B 0,C 180,E1 26279.17,E2 26279.17} C_VEL
LIN {X 0,Y 551.916,Z 1158.886,A -85,B 0,C 180,E1 26277.508,E2 26277.508} C_VEL
LIN {X 0,Y 551.916,Z 1156.725,A -85,B 0,C 180,E1 26275.741,E2 26275.741} C_VEL
LIN {X 0,Y 551.932,Z 1152.732,A -85,B 0,C 180,E1 26273.969,E2 26273.969} C_VEL
LIN {X 0,Y 551.963,Z 1147.672,A -85,B 0,C 180,E1 26272.401,E2 26272.401} C_VEL
LIN {X 0,Y 552.044,Z 1140.557,A -85,B 0,C 180,E1 26270.724,E2 26270.724} C_VEL
LIN {X 0,Y 552.174,Z 1131.29,A -85,B 0,C 180,E1 26269.04,E2 26269.04} C_VEL
LIN {X 0,Y 552.332,Z 1121.888,A -85,B 0,C 180,E1 26267.666,E2 26267.666} C_VEL
LIN {X 0,Y 552.567,Z 1110.54,A -85,B 0,C 180,E1 26266.288,E2 26266.288} C_VEL
LIN {X 0,Y 552.869,Z 1097.048,A -85,B 0,C 180,E1 26264.958,E2 26264.958} C_VEL
LIN {X 0,Y 553.163,Z 1083.784,A -85,B 0,C 180,E1 26263.892,E2 26263.892} C_VEL
LIN {X 0,Y 553.495,Z 1069.227,A -85,B 0,C 180,E1 26262.93,E2 26262.93} C_VEL
LIN {X 0,Y 553.816,Z 1052.574,A -85,B 0,C 180,E1 26262.073,E2 26262.073} C_VEL
LIN {X 0,Y 554.074,Z 1037.451,A -85,B 0,C 180,E1 26261.482,E2 26261.482} C_VEL
LIN {X 0,Y 554.306,Z 1020.866,A -85,B 0,C 180,E1 26261.013,E2 26261.013} C_VEL
LIN {X 0,Y 554.456,Z 998.776,A -85,B 0,C 180,E1 26260.652,E2 26260.652} C_VEL
LIN {X 0,Y 554.811,Z 849.919,A -85,B 0,C 180,E1 26258.665,E2 26258.665} C_VEL
LIN {X 0,Y 554.074,Z 844.749,A -85,B 0,C 180,E1 26258.561,E2 26258.561} C_VEL
LIN {X 0,Y 554.832,Z 801.645,A -85,B 0,C 180,E1 26255.173,E2 26255.173} C_VEL
LIN {X 0,Y 555.712,Z 760.706,A -85,B 0,C 180,E1 26251.875,E2 26251.875} C_VEL
LIN {X 0,Y 558.885,Z 732.347,A -85,B 0,C 180,E1 26249.047,E2 26249.047} C_VEL
LIN {X 0,Y 562.785,Z 710.214,A -85,B 0,C 180,E1 26246.703,E2 26246.703} C_VEL
LIN {X 0,Y 567.658,Z 692.446,A -85,B 0,C 180,E1 26244.606,E2 26244.606} C_VEL
LIN {X 0,Y 566.578,Z 689.896,A -85,B 0,C 180,E1 26243.075,E2 26243.075} C_VEL
LIN {X 0,Y 566.738,Z 689.518,A -85,B 0,C 180,E1 26242.221,E2 26242.221} C_VEL
LIN {X 0,Y 566.736,Z 690.037,A -85,B 0,C 180,E1 26241.893,E2 26241.893} C_VEL
LIN {X 0,Y 562.394,Z 700.4,A -85,B 0,C 180,E1 26240.98,E2 26240.98} C_VEL
LIN {X 0,Y 559.45,Z 712.419,A -85,B 0,C 180,E1 26240.06,E2 26240.06} C_VEL
LIN {X 0,Y 557.389,Z 729.628,A -85,B 0,C 180,E1 26238.93,E2 26238.93} C_VEL
LIN {X 0,Y 556.817,Z 750.626,A -85,B 0,C 180,E1 26237.672,E2 26237.672} C_VEL
LIN {X 0,Y 558.272,Z 768.047,A -85,B 0,C 180,E1 26236.627,E2 26236.627} C_VEL
LIN {X 0,Y 561.326,Z 781.229,A -85,B 0,C 180,E1 26235.785,E2 26235.785} C_VEL
LIN {X 0,Y 565.615,Z 791.552,A -85,B 0,C 180,E1 26235.073,E2 26235.073} C_VEL
LIN {X 0,Y 571.225,Z 800.083,A -85,B 0,C 180,E1 26234.427,E2 26234.427} C_VEL
LIN {X 0,Y 577.917,Z 806.908,A -85,B 0,C 180,E1 26233.826,E2 26233.826} C_VEL
LIN {X 0,Y 582.171,Z 809.968,A -85,B 0,C 180,E1 26233.408,E2 26233.408} C_VEL
LIN {X 0,Y 585.781,Z 811.705,A -85,B 0,C 180,E1 26232.925,E2 26232.925} C_VEL
LIN {X 0,Y 588.693,Z 812.232,A -85,B 0,C 180,E1 26232.369,E2 26232.369} C_VEL
LIN {X 0,Y 590.43,Z 811.651,A -85,B 0,C 180,E1 26231.831,E2 26231.831} C_VEL
LIN {X 0,Y 591.15,Z 809.876,A -85,B 0,C 180,E1 26231.226,E2 26231.226} C_VEL
LIN {X 0,Y 590.468,Z 806.954,A -85,B 0,C 180,E1 26230.646,E2 26230.646} C_VEL
LIN {X 0,Y 588.382,Z 803.048,A -85,B 0,C 180,E1 26230.142,E2 26230.142} C_VEL
LIN {X 0,Y 583.582,Z 795.63,A -85,B 0,C 180,E1 26229.547,E2 26229.547} C_VEL
LIN {X 0,Y 579.23,Z 786.372,A -85,B 0,C 180,E1 26229.023,E2 26229.023} C_VEL
LIN {X 0,Y 575.861,Z 775.781,A -85,B 0,C 180,E1 26228.607,E2 26228.607} C_VEL
LIN {X 0,Y 573.49,Z 763.753,A -85,B 0,C 180,E1 26228.31,E2 26228.31} C_VEL
LIN {X 0,Y 572.118,Z 749.858,A -85,B 0,C 180,E1 26228.136,E2 26228.136} C_VEL
LIN {X 0,Y 571.773,Z 731.56,A -85,B 0,C 180,E1 26228.092,E2 26228.092} C_VEL
LIN {X 0,Y 571.751,Z 725.675,A -85,B 0,C 180,E1 26228.089,E2 26228.089} C_VEL
LIN {X 0,Y 570.174,Z 727.028,A -85,B 0,C 180,E1 26227.886,E2 26227.886} C_VEL
LIN {X 0,Y 566.168,Z 736.676,A -85,B 0,C 180,E1 26227.362,E2 26227.362} C_VEL
LIN {X 0,Y 562.923,Z 741.971,A -85,B 0,C 180,E1 26226.927,E2 26226.927} C_VEL
LIN {X 0,Y 560.977,Z 743.526,A -85,B 0,C 180,E1 26226.662,E2 26226.662} C_VEL
LIN {X 0,Y 559.951,Z 743.382,A -85,B 0,C 180,E1 26226.517,E2 26226.517} C_VEL
LIN {X 0,Y 559.698,Z 759.562,A -85,B 0,C 180,E1 26225.551,E2 26225.551} C_VEL
LIN {X 0,Y 561.192,Z 770.091,A -85,B 0,C 180,E1 26225.28,E2 26225.28} C_VEL
LIN {X 0,Y 559.52,Z 1004.969,A -85,B 0,C 180,E1 26221.854,E2 26221.854} C_VEL
LIN {X 0,Y 559.035,Z 1066.253,A -85,B 0,C 180,E1 26220.945,E2 26220.945} C_VEL
LIN {X 0,Y 558.589,Z 1088.478,A -85,B 0,C 180,E1 26220.418,E2 26220.418} C_VEL
LIN {X 0,Y 558.03,Z 1110.457,A -85,B 0,C 180,E1 26219.692,E2 26219.692} C_VEL
LIN {X 0,Y 557.4,Z 1131.557,A -85,B 0,C 180,E1 26218.792,E2 26218.792} C_VEL
LIN {X 0,Y 556.677,Z 1151.764,A -85,B 0,C 180,E1 26217.723,E2 26217.723} C_VEL
LIN {X 0,Y 555.937,Z 1171.647,A -85,B 0,C 180,E1 26216.455,E2 26216.455} C_VEL
LIN {X 0,Y 555.19,Z 1190.466,A -85,B 0,C 180,E1 26215.038,E2 26215.038} C_VEL
LIN {X 0,Y 554.497,Z 1208.057,A -85,B 0,C 180,E1 26213.485,E2 26213.485} C_VEL
LIN {X 0,Y 553.887,Z 1224.188,A -85,B 0,C 180,E1 26211.831,E2 26211.831} C_VEL
LIN {X 0,Y 553.296,Z 1240.74,A -85,B 0,C 180,E1 26209.861,E2 26209.861} C_VEL
LIN {X 0,Y 552.849,Z 1254.758,A -85,B 0,C 180,E1 26207.906,E2 26207.906} C_VEL
LIN {X 0,Y 552.492,Z 1267.336,A -85,B 0,C 180,E1 26205.859,E2 26205.859} C_VEL
LIN {X 0,Y 552.242,Z 1278.365,A -85,B 0,C 180,E1 26203.721,E2 26203.721} C_VEL
LIN {X 0,Y 552.081,Z 1287.717,A -85,B 0,C 180,E1 26201.54,E2 26201.54} C_VEL
LIN {X 0,Y 551.985,Z 1295.535,A -85,B 0,C 180,E1 26199.278,E2 26199.278} C_VEL
LIN {X 0,Y 551.932,Z 1301.155,A -85,B 0,C 180,E1 26197.181,E2 26197.181} C_VEL
LIN {X 0,Y 551.907,Z 1305.672,A -85,B 0,C 180,E1 26194.864,E2 26194.864} C_VEL
LIN {X 0,Y 551.9,Z 1308.392,A -85,B 0,C 180,E1 26192.596,E2 26192.596} C_VEL
LIN {X 0,Y 551.894,Z 1309.395,A -85,B 0,C 180,E1 26190.519,E2 26190.519} C_VEL
LIN {X 0,Y 551.9,Z 1308.896,A -85,B 0,C 180,E1 26188.132,E2 26188.132} C_VEL
LIN {X 0,Y 551.903,Z 1306.849,A -85,B 0,C 180,E1 26185.949,E2 26185.949} C_VEL
LIN {X 0,Y 551.911,Z 1303.408,A -85,B 0,C 180,E1 26183.865,E2 26183.865} C_VEL
LIN {X 0,Y 551.954,Z 1297.984,A -85,B 0,C 180,E1 26181.563,E2 26181.563} C_VEL
LIN {X 0,Y 552.022,Z 1291.412,A -85,B 0,C 180,E1 26179.46,E2 26179.46} C_VEL
LIN {X 0,Y 552.156,Z 1282.7,A -85,B 0,C 180,E1 26177.237,E2 26177.237} C_VEL
LIN {X 0,Y 552.36,Z 1272.537,A -85,B 0,C 180,E1 26175.106,E2 26175.106} C_VEL
LIN {X 0,Y 552.651,Z 1261.466,A -85,B 0,C 180,E1 26173.149,E2 26173.149} C_VEL
LIN {X 0,Y 553.06,Z 1248.041,A -85,B 0,C 180,E1 26171.119,E2 26171.119} C_VEL
LIN {X 0,Y 553.571,Z 1232.803,A -85,B 0,C 180,E1 26169.157,E2 26169.157} C_VEL
LIN {X 0,Y 554.166,Z 1217.035,A -85,B 0,C 180,E1 26167.4,E2 26167.4} C_VEL
LIN {X 0,Y 554.876,Z 1198.387,A -85,B 0,C 180,E1 26165.629,E2 26165.629} C_VEL
LIN {X 0,Y 555.617,Z 1179.776,A -85,B 0,C 180,E1 26164.128,E2 26164.128} C_VEL
LIN {X 0,Y 556.38,Z 1160.107,A -85,B 0,C 180,E1 26162.782,E2 26162.782} C_VEL
LIN {X 0,Y 557.091,Z 1139.435,A -85,B 0,C 180,E1 26161.601,E2 26161.601} C_VEL
LIN {X 0,Y 557.817,Z 1118.221,A -85,B 0,C 180,E1 26160.615,E2 26160.615} C_VEL
LIN {X 0,Y 558.39,Z 1096.975,A -85,B 0,C 180,E1 26159.84,E2 26159.84} C_VEL
LIN {X 0,Y 558.874,Z 1075.089,A -85,B 0,C 180,E1 26159.24,E2 26159.24} C_VEL
LIN {X 0,Y 559.198,Z 1052.373,A -85,B 0,C 180,E1 26158.825,E2 26158.825} C_VEL
LIN {X 0,Y 560.763,Z 826.401,A -85,B 0,C 180,E1 26155.55,E2 26155.55} C_VEL
LIN {X 0,Y 561.013,Z 767.546,A -85,B 0,C 180,E1 26154.668,E2 26154.668} C_VEL
LIN {X 0,Y 559.596,Z 758.121,A -85,B 0,C 180,E1 26154.387,E2 26154.387} C_VEL
LIN {X 0,Y 560.077,Z 743.406,A -85,B 0,C 180,E1 26153.462,E2 26153.462} C_VEL
LIN {X 0,Y 561.57,Z 743.246,A -85,B 0,C 180,E1 26153.257,E2 26153.257} C_VEL
LIN {X 0,Y 564.197,Z 740.199,A -85,B 0,C 180,E1 26152.901,E2 26152.901} C_VEL
LIN {X 0,Y 567.988,Z 732.709,A -85,B 0,C 180,E1 26152.398,E2 26152.398} C_VEL
LIN {X 0,Y 570.361,Z 726.646,A -85,B 0,C 180,E1 26152.09,E2 26152.09} C_VEL
LIN {X 0,Y 571.77,Z 725.66,A -85,B 0,C 180,E1 26151.909,E2 26151.909} C_VEL
LIN {X 0,Y 572.045,Z 748.479,A -85,B 0,C 180,E1 26151.874,E2 26151.874} C_VEL
LIN {X 0,Y 573.33,Z 762.622,A -85,B 0,C 180,E1 26151.71,E2 26151.71} C_VEL
LIN {X 0,Y 575.622,Z 774.813,A -85,B 0,C 180,E1 26151.422,E2 26151.422} C_VEL
LIN {X 0,Y 578.909,Z 785.526,A -85,B 0,C 180,E1 26151.016,E2 26151.016} C_VEL
LIN {X 0,Y 583.179,Z 794.896,A -85,B 0,C 180,E1 26150.501,E2 26150.501} C_VEL
LIN {X 0,Y 588.106,Z 802.614,A -85,B 0,C 180,E1 26149.901,E2 26149.901} C_VEL
LIN {X 0,Y 590.275,Z 806.497,A -85,B 0,C 180,E1 26149.425,E2 26149.425} C_VEL
LIN {X 0,Y 591.142,Z 809.538,A -85,B 0,C 180,E1 26148.857,E2 26148.857} C_VEL
LIN {X 0,Y 590.677,Z 811.393,A -85,B 0,C 180,E1 26148.287,E2 26148.287} C_VEL
LIN {X 0,Y 589.094,Z 812.21,A -85,B 0,C 180,E1 26147.732,E2 26147.732} C_VEL
LIN {X 0,Y 586.318,Z 811.878,A -85,B 0,C 180,E1 26147.162,E2 26147.162} C_VEL
LIN {X 0,Y 582.818,Z 810.341,A -85,B 0,C 180,E1 26146.668,E2 26146.668} C_VEL
LIN {X 0,Y 576.585,Z 805.76,A -85,B 0,C 180,E1 26145.883,E2 26145.883} C_VEL
LIN {X 0,Y 571.656,Z 799.936,A -85,B 0,C 180,E1 26145.102,E2 26145.102} C_VEL
LIN {X 0,Y 567.594,Z 791.99,A -85,B 0,C 180,E1 26144.233,E2 26144.233} C_VEL
LIN {X 0,Y 564.872,Z 782.186,A -85,B 0,C 180,E1 26143.324,E2 26143.324} C_VEL
LIN {X 0,Y 563.479,Z 769.723,A -85,B 0,C 180,E1 26142.323,E2 26142.323} C_VEL
LIN {X 0,Y 563.658,Z 750.495,A -85,B 0,C 180,E1 26140.971,E2 26140.971} C_VEL
LIN {X 0,Y 565.007,Z 712.592,A -85,B 0,C 180,E1 26138.335,E2 26138.335} C_VEL
LIN {X 0,Y 565.809,Z 691.579,A -85,B 0,C 180,E1 26136.802,E2 26136.802} C_VEL
LIN {X 0,Y 559.216,Z 679.296,A -85,B 0,C 180,E1 26135.025,E2 26135.025} C_VEL
LIN {X 0,Y 557.101,Z 675.254,A -85,B 0,C 180,E1 26134.426,E2 26134.426} C_VEL
LIN {X 0,Y 554.987,Z 671.25,A -85,B 0,C 180,E1 26133.827,E2 26133.827} C_VEL
LIN {X 0,Y 552.76,Z 667.679,A -85,B 0,C 180,E1 26133.235,E2 26133.235} C_VEL
LIN {X 0,Y 552.343,Z 665.937,A -85,B 0,C 180,E1 26133.016,E2 26133.016} C_VEL
LIN {X 0,Y 552.337,Z 665.935,A -85,B 0,C 180,E1 26129.497,E2 26129.497} C_VEL
LIN {X 0,Y 552.342,Z 665.932,A -85,B 0,C 180,E1 26126.096,E2 26126.096} C_VEL
LIN {X 0,Y 552.342,Z 665.935,A -85,B 0,C 180,E1 26122.679,E2 26122.679} C_VEL
LIN {X 0,Y 552.326,Z 665.935,A -85,B 0,C 180,E1 26119.346,E2 26119.346} C_VEL
LIN {X 0,Y 552.331,Z 665.934,A -85,B 0,C 180,E1 26116.006,E2 26116.006} C_VEL
LIN {X 0,Y 552.33,Z 665.934,A -85,B 0,C 180,E1 26112.652,E2 26112.652} C_VEL
LIN {X 0,Y 552.338,Z 665.934,A -85,B 0,C 180,E1 26109.271,E2 26109.271} C_VEL
LIN {X 0,Y 552.341,Z 665.934,A -85,B 0,C 180,E1 26105.922,E2 26105.922} C_VEL
LIN {X 0,Y 552.336,Z 665.936,A -85,B 0,C 180,E1 26102.594,E2 26102.594} C_VEL
LIN {X 0,Y 552.333,Z 665.935,A -85,B 0,C 180,E1 26099.274,E2 26099.274} C_VEL
LIN {X 0,Y 552.327,Z 665.933,A -85,B 0,C 180,E1 26095.902,E2 26095.902} C_VEL
LIN {X 0,Y 552.325,Z 665.934,A -85,B 0,C 180,E1 26092.615,E2 26092.615} C_VEL
LIN {X 0,Y 552.33,Z 665.934,A -85,B 0,C 180,E1 26089.254,E2 26089.254} C_VEL
LIN {X 0,Y 552.327,Z 665.935,A -85,B 0,C 180,E1 26085.961,E2 26085.961} C_VEL
LIN {X 0,Y 552.34,Z 665.937,A -85,B 0,C 180,E1 26082.621,E2 26082.621} C_VEL
LIN {X 0,Y 552.344,Z 665.934,A -85,B 0,C 180,E1 26079.219,E2 26079.219} C_VEL
LIN {X 0,Y 552.339,Z 665.931,A -85,B 0,C 180,E1 26075.737,E2 26075.737} C_VEL
LIN {X 0,Y 552.337,Z 665.926,A -85,B 0,C 180,E1 26072.715,E2 26072.715} C_VEL
LIN {X 0,Y 551.367,Z 666.046,A -85,B 0,C 180,E1 26071.916,E2 26071.916} C_VEL
LIN {X 0,Y 544.849,Z 666.86,A -85,B 0,C 180,E1 26069.614,E2 26069.614} C_VEL
LIN {X 0,Y 544.397,Z 666.918,A -85,B 0,C 180,E1 26069.088,E2 26069.088} C_VEL
LIN {X 0,Y 544.399,Z 666.913,A -85,B 0,C 180,E1 26065.678,E2 26065.678} C_VEL
LIN {X 0,Y 544.397,Z 666.925,A -85,B 0,C 180,E1 26062.294,E2 26062.294} C_VEL
LIN {X 0,Y 544.386,Z 666.912,A -85,B 0,C 180,E1 26059.013,E2 26059.013} C_VEL
LIN {X 0,Y 544.386,Z 666.924,A -85,B 0,C 180,E1 26055.738,E2 26055.738} C_VEL
LIN {X 0,Y 544.389,Z 666.927,A -85,B 0,C 180,E1 26052.38,E2 26052.38} C_VEL
LIN {X 0,Y 544.393,Z 666.93,A -85,B 0,C 180,E1 26049.022,E2 26049.022} C_VEL
LIN {X 0,Y 544.395,Z 666.993,A -85,B 0,C 180,E1 26048.239,E2 26048.239} C_VEL
LIN {X 0,Y 545.328,Z 669.801,A -85,B 0,C 180,E1 26047.963,E2 26047.963} C_VEL
LIN {X 0,Y 552.245,Z 686.603,A -85,B 0,C 180,E1 26046.244,E2 26046.244} C_VEL
LIN {X 0,Y 551.139,Z 731.622,A -85,B 0,C 180,E1 26043.159,E2 26043.159} C_VEL
LIN {X 0,Y 550.261,Z 766.147,A -85,B 0,C 180,E1 26040.833,E2 26040.833} C_VEL
LIN {X 0,Y 551.829,Z 776.98,A -85,B 0,C 180,E1 26040.575,E2 26040.575} C_VEL
LIN {X 0,Y 550.228,Z 1012.33,A -85,B 0,C 180,E1 26037.233,E2 26037.233} C_VEL
LIN {X 0,Y 549.931,Z 1035.56,A -85,B 0,C 180,E1 26036.826,E2 26036.826} C_VEL
LIN {X 0,Y 549.484,Z 1056.274,A -85,B 0,C 180,E1 26036.263,E2 26036.263} C_VEL
LIN {X 0,Y 548.944,Z 1076.29,A -85,B 0,C 180,E1 26035.516,E2 26035.516} C_VEL
LIN {X 0,Y 548.331,Z 1095.005,A -85,B 0,C 180,E1 26034.623,E2 26034.623} C_VEL
LIN {X 0,Y 547.648,Z 1113.85,A -85,B 0,C 180,E1 26033.51,E2 26033.51} C_VEL
LIN {X 0,Y 546.99,Z 1131.014,A -85,B 0,C 180,E1 26032.289,E2 26032.289} C_VEL
LIN {X 0,Y 546.32,Z 1148.057,A -85,B 0,C 180,E1 26030.852,E2 26030.852} C_VEL
LIN {X 0,Y 545.705,Z 1164.063,A -85,B 0,C 180,E1 26029.256,E2 26029.256} C_VEL
LIN {X 0,Y 545.164,Z 1178.951,A -85,B 0,C 180,E1 26027.502,E2 26027.502} C_VEL
LIN {X 0,Y 544.739,Z 1192.209,A -85,B 0,C 180,E1 26025.653,E2 26025.653} C_VEL
LIN {X 0,Y 544.407,Z 1204.006,A -85,B 0,C 180,E1 26023.696,E2 26023.696} C_VEL
LIN {X 0,Y 544.179,Z 1214.193,A -85,B 0,C 180,E1 26021.66,E2 26021.66} C_VEL
LIN {X 0,Y 544.039,Z 1222.417,A -85,B 0,C 180,E1 26019.627,E2 26019.627} C_VEL
LIN {X 0,Y 543.965,Z 1228.883,A -85,B 0,C 180,E1 26017.604,E2 26017.604} C_VEL
LIN {X 0,Y 543.922,Z 1234.173,A -85,B 0,C 180,E1 26015.379,E2 26015.379} C_VEL
LIN {X 0,Y 543.913,Z 1237.507,A -85,B 0,C 180,E1 26013.266,E2 26013.266} C_VEL
LIN {X 0,Y 543.91,Z 1239.242,A -85,B 0,C 180,E1 26011.158,E2 26011.158} C_VEL
LIN {X 0,Y 543.912,Z 1239.316,A -85,B 0,C 180,E1 26009.052,E2 26009.052} C_VEL
LIN {X 0,Y 543.915,Z 1237.828,A -85,B 0,C 180,E1 26006.944,E2 26006.944} C_VEL
LIN {X 0,Y 543.918,Z 1234.55,A -85,B 0,C 180,E1 26004.726,E2 26004.726} C_VEL
LIN {X 0,Y 543.944,Z 1230.035,A -85,B 0,C 180,E1 26002.713,E2 26002.713} C_VEL
LIN {X 0,Y 544.018,Z 1223.505,A -85,B 0,C 180,E1 26000.585,E2 26000.585} C_VEL
LIN {X 0,Y 544.159,Z 1215.498,A -85,B 0,C 180,E1 25998.554,E2 25998.554} C_VEL
LIN {X 0,Y 544.37,Z 1205.592,A -85,B 0,C 180,E1 25996.51,E2 25996.51} C_VEL
LIN {X 0,Y 544.686,Z 1193.911,A -85,B 0,C 180,E1 25994.52,E2 25994.52} C_VEL
LIN {X 0,Y 545.118,Z 1180.449,A -85,B 0,C 180,E1 25992.604,E2 25992.604} C_VEL
LIN {X 0,Y 545.657,Z 1165.365,A -85,B 0,C 180,E1 25990.797,E2 25990.797} C_VEL
LIN {X 0,Y 546.263,Z 1149.606,A -85,B 0,C 180,E1 25989.201,E2 25989.201} C_VEL
LIN {X 0,Y 546.918,Z 1132.871,A -85,B 0,C 180,E1 25987.763,E2 25987.763} C_VEL
LIN {X 0,Y 547.602,Z 1115.228,A -85,B 0,C 180,E1 25986.487,E2 25986.487} C_VEL
LIN {X 0,Y 548.281,Z 1096.605,A -85,B 0,C 180,E1 25985.373,E2 25985.373} C_VEL
LIN {X 0,Y 548.872,Z 1078.24,A -85,B 0,C 180,E1 25984.48,E2 25984.48} C_VEL
LIN {X 0,Y 549.44,Z 1057.658,A -85,B 0,C 180,E1 25983.693,E2 25983.693} C_VEL
LIN {X 0,Y 549.91,Z 1036.836,A -85,B 0,C 180,E1 25983.113,E2 25983.113} C_VEL
LIN {X 0,Y 550.215,Z 1014.4,A -85,B 0,C 180,E1 25982.706,E2 25982.706} C_VEL
LIN {X 0,Y 551.81,Z 780.056,A -85,B 0,C 180,E1 25979.38,E2 25979.38} C_VEL
LIN {X 0,Y 548.971,Z 767.43,A -85,B 0,C 180,E1 25978.999,E2 25978.999} C_VEL
LIN {X 0,Y 550.106,Z 732.825,A -85,B 0,C 180,E1 25975.607,E2 25975.607} C_VEL
LIN {X 0,Y 550.98,Z 699.27,A -85,B 0,C 180,E1 25972.298,E2 25972.298} C_VEL
LIN {X 0,Y 551.084,Z 685.821,A -85,B 0,C 180,E1 25970.945,E2 25970.945} C_VEL
LIN {X 0,Y 545.265,Z 669.682,A -85,B 0,C 180,E1 25968.829,E2 25968.829} C_VEL
LIN {X 0,Y 544.386,Z 666.927,A -85,B 0,C 180,E1 25968.468,E2 25968.468} C_VEL
LIN {X 0,Y 544.387,Z 666.923,A -85,B 0,C 180,E1 25965.147,E2 25965.147} C_VEL
LIN {X 0,Y 544.4,Z 666.924,A -85,B 0,C 180,E1 25961.783,E2 25961.783} C_VEL
LIN {X 0,Y 544.4,Z 666.923,A -85,B 0,C 180,E1 25958.349,E2 25958.349} C_VEL
LIN {X 0,Y 544.424,Z 667.128,A -85,B 0,C 180,E1 25955.188,E2 25955.188} C_VEL
LIN {X 0,Y 551.192,Z 685.283,A -85,B 0,C 180,E1 25952.97,E2 25952.97} C_VEL
LIN {X 0,Y 549.744,Z 724.864,A -85,B 0,C 180,E1 25949.531,E2 25949.531} C_VEL
LIN {X 0,Y 548.326,Z 765.471,A -85,B 0,C 180,E1 25946.07,E2 25946.07} C_VEL
LIN {X 0,Y 547.438,Z 796.16,A -85,B 0,C 180,E1 25943.527,E2 25943.527} C_VEL
LIN {X 0,Y 546.53,Z 839.509,A -85,B 0,C 180,E1 25940.061,E2 25940.061} C_VEL
LIN {X 0,Y 546.475,Z 845.247,A -85,B 0,C 180,E1 25939.633,E2 25939.633} C_VEL
LIN {X 0,Y 547.491,Z 854.187,A -85,B 0,C 180,E1 25939.47,E2 25939.47} C_VEL
LIN {X 0,Y 546.74,Z 1014.374,A -85,B 0,C 180,E1 25937.285,E2 25937.285} C_VEL
LIN {X 0,Y 546.537,Z 1031.689,A -85,B 0,C 180,E1 25936.871,E2 25936.871} C_VEL
LIN {X 0,Y 546.22,Z 1048.36,A -85,B 0,C 180,E1 25936.264,E2 25936.264} C_VEL
LIN {X 0,Y 545.901,Z 1062.655,A -85,B 0,C 180,E1 25935.58,E2 25935.58} C_VEL
LIN {X 0,Y 545.528,Z 1078.076,A -85,B 0,C 180,E1 25934.651,E2 25934.651} C_VEL
LIN {X 0,Y 545.143,Z 1092.763,A -85,B 0,C 180,E1 25933.53,E2 25933.53} C_VEL
LIN {X 0,Y 544.822,Z 1104.925,A -85,B 0,C 180,E1 25932.399,E2 25932.399} C_VEL
LIN {X 0,Y 544.542,Z 1116.471,A -85,B 0,C 180,E1 25931.116,E2 25931.116} C_VEL
LIN {X 0,Y 544.28,Z 1128.114,A -85,B 0,C 180,E1 25929.517,E2 25929.517} C_VEL
LIN {X 0,Y 544.116,Z 1136.864,A -85,B 0,C 180,E1 25928.028,E2 25928.028} C_VEL
LIN {X 0,Y 544.012,Z 1144.446,A -85,B 0,C 180,E1 25926.437,E2 25926.437} C_VEL
LIN {X 0,Y 543.947,Z 1150.926,A -85,B 0,C 180,E1 25924.639,E2 25924.639} C_VEL
LIN {X 0,Y 543.919,Z 1155.276,A -85,B 0,C 180,E1 25922.951,E2 25922.951} C_VEL
LIN {X 0,Y 543.912,Z 1158.232,A -85,B 0,C 180,E1 25921.159,E2 25921.159} C_VEL
LIN {X 0,Y 543.915,Z 1159.443,A -85,B 0,C 180,E1 25919.263,E2 25919.263} C_VEL
LIN {X 0,Y 543.915,Z 1158.944,A -85,B 0,C 180,E1 25917.577,E2 25917.577} C_VEL
LIN {X 0,Y 543.917,Z 1157.014,A -85,B 0,C 180,E1 25915.889,E2 25915.889} C_VEL
LIN {X 0,Y 543.934,Z 1152.942,A -85,B 0,C 180,E1 25913.97,E2 25913.97} C_VEL
LIN {X 0,Y 543.973,Z 1147.608,A -85,B 0,C 180,E1 25912.289,E2 25912.289} C_VEL
LIN {X 0,Y 544.06,Z 1140.971,A -85,B 0,C 180,E1 25910.693,E2 25910.693} C_VEL
LIN {X 0,Y 544.22,Z 1131.182,A -85,B 0,C 180,E1 25908.878,E2 25908.878} C_VEL
LIN {X 0,Y 544.41,Z 1121.763,A -85,B 0,C 180,E1 25907.484,E2 25907.484} C_VEL
LIN {X 0,Y 544.658,Z 1111.327,A -85,B 0,C 180,E1 25906.193,E2 25906.193} C_VEL
LIN {X 0,Y 545.024,Z 1097.445,A -85,B 0,C 180,E1 25904.788,E2 25904.788} C_VEL
LIN {X 0,Y 545.359,Z 1084.287,A -85,B 0,C 180,E1 25903.71,E2 25903.71} C_VEL
LIN {X 0,Y 545.713,Z 1070.721,A -85,B 0,C 180,E1 25902.789,E2 25902.789} C_VEL
LIN {X 0,Y 546.113,Z 1053.432,A -85,B 0,C 180,E1 25901.866,E2 25901.866} C_VEL
LIN {X 0,Y 546.411,Z 1038.086,A -85,B 0,C 180,E1 25901.252,E2 25901.252} C_VEL
LIN {X 0,Y 546.65,Z 1022.731,A -85,B 0,C 180,E1 25900.802,E2 25900.802} C_VEL
LIN {X 0,Y 546.84,Z 1003.813,A -85,B 0,C 180,E1 25900.457,E2 25900.457} C_VEL
LIN {X 0,Y 547.291,Z 850.752,A -85,B 0,C 180,E1 25898.385,E2 25898.385} C_VEL
LIN {X 0,Y 546.434,Z 844.516,A -85,B 0,C 180,E1 25898.244,E2 25898.244} C_VEL
LIN {X 0,Y 547.301,Z 802.141,A -85,B 0,C 180,E1 25894.865,E2 25894.865} C_VEL
LIN {X 0,Y 547.818,Z 784.229,A -85,B 0,C 180,E1 25893.38,E2 25893.38} C_VEL
LIN {X 0,Y 550.434,Z 757.15,A -85,B 0,C 180,E1 25890.749,E2 25890.749} C_VEL
LIN {X 0,Y 553.416,Z 735.242,A -85,B 0,C 180,E1 25888.514,E2 25888.514} C_VEL
LIN {X 0,Y 557.954,Z 713.483,A -85,B 0,C 180,E1 25886.13,E2 25886.13} C_VEL
LIN {X 0,Y 562.722,Z 698.465,A -85,B 0,C 180,E1 25884.293,E2 25884.293} C_VEL
LIN {X 0,Y 562.149,Z 696.417,A -85,B 0,C 180,E1 25882.918,E2 25882.918} C_VEL
LIN {X 0,Y 562.298,Z 696.23,A -85,B 0,C 180,E1 25882.306,E2 25882.306} C_VEL
LIN {X 0,Y 556.838,Z 707.317,A -85,B 0,C 180,E1 25881.278,E2 25881.278} C_VEL
LIN {X 0,Y 553.373,Z 718.885,A -85,B 0,C 180,E1 25880.329,E2 25880.329} C_VEL
LIN {X 0,Y 550.947,Z 733.912,A -85,B 0,C 180,E1 25879.26,E2 25879.26} C_VEL
LIN {X 0,Y 549.981,Z 752.853,A -85,B 0,C 180,E1 25878.036,E2 25878.036} C_VEL
LIN {X 0,Y 551.028,Z 769.439,A -85,B 0,C 180,E1 25876.98,E2 25876.98} C_VEL
LIN {X 0,Y 553.723,Z 782.713,A -85,B 0,C 180,E1 25876.094,E2 25876.094} C_VEL
LIN {X 0,Y 557.928,Z 793.884,A -85,B 0,C 180,E1 25875.3,E2 25875.3} C_VEL
LIN {X 0,Y 563.244,Z 802.825,A -85,B 0,C 180,E1 25874.615,E2 25874.615} C_VEL
LIN {X 0,Y 569.705,Z 810.252,A -85,B 0,C 180,E1 25873.981,E2 25873.981} C_VEL
LIN {X 0,Y 576.715,Z 815.932,A -85,B 0,C 180,E1 25873.413,E2 25873.413} C_VEL
LIN {X 0,Y 581.243,Z 818.396,A -85,B 0,C 180,E1 25872.938,E2 25872.938} C_VEL
LIN {X 0,Y 584.866,Z 819.442,A -85,B 0,C 180,E1 25872.394,E2 25872.394} C_VEL
LIN {X 0,Y 587.422,Z 819.23,A -85,B 0,C 180,E1 25871.796,E2 25871.796} C_VEL
LIN {X 0,Y 588.675,Z 817.86,A -85,B 0,C 180,E1 25871.199,E2 25871.199} C_VEL
LIN {X 0,Y 588.559,Z 815.324,A -85,B 0,C 180,E1 25870.591,E2 25870.591} C_VEL
LIN {X 0,Y 586.986,Z 811.881,A -85,B 0,C 180,E1 25870.05,E2 25870.05} C_VEL
LIN {X 0,Y 583.98,Z 807.479,A -85,B 0,C 180,E1 25869.594,E2 25869.594} C_VEL
LIN {X 0,Y 578.837,Z 799.163,A -85,B 0,C 180,E1 25868.975,E2 25868.975} C_VEL
LIN {X 0,Y 574.421,Z 789.105,A -85,B 0,C 180,E1 25868.427,E2 25868.427} C_VEL
LIN {X 0,Y 571.019,Z 777.789,A -85,B 0,C 180,E1 25867.995,E2 25867.995} C_VEL
LIN {X 0,Y 568.623,Z 765.079,A -85,B 0,C 180,E1 25867.685,E2 25867.685} C_VEL
LIN {X 0,Y 567.232,Z 750.577,A -85,B 0,C 180,E1 25867.502,E2 25867.502} C_VEL
LIN {X 0,Y 566.928,Z 746.908,A -85,B 0,C 180,E1 25867.462,E2 25867.462} C_VEL
LIN {X 0,Y 563.675,Z 750.451,A -85,B 0,C 180,E1 25867.029,E2 25867.029} C_VEL
LIN {X 0,Y 562.811,Z 751.36,A -85,B 0,C 180,E1 25866.912,E2 25866.912} C_VEL
LIN {X 0,Y 558.746,Z 761.529,A -85,B 0,C 180,E1 25866.354,E2 25866.354} C_VEL
LIN {X 0,Y 556.458,Z 768.091,A -85,B 0,C 180,E1 25866.032,E2 25866.032} C_VEL
LIN {X 0,Y 555.066,Z 769.72,A -85,B 0,C 180,E1 25865.834,E2 25865.834} C_VEL
LIN {X 0,Y 554.636,Z 769.978,A -85,B 0,C 180,E1 25865.762,E2 25865.762} C_VEL
LIN {X 0,Y 552.833,Z 990.855,A -85,B 0,C 180,E1 25862.498,E2 25862.498} C_VEL
LIN {X 0,Y 552.177,Z 1065.887,A -85,B 0,C 180,E1 25861.38,E2 25861.38} C_VEL
LIN {X 0,Y 551.658,Z 1088.132,A -85,B 0,C 180,E1 25860.852,E2 25860.852} C_VEL
LIN {X 0,Y 551.031,Z 1110.314,A -85,B 0,C 180,E1 25860.114,E2 25860.114} C_VEL
LIN {X 0,Y 550.289,Z 1131.552,A -85,B 0,C 180,E1 25859.2,E2 25859.2} C_VEL
LIN {X 0,Y 549.469,Z 1151.771,A -85,B 0,C 180,E1 25858.119,E2 25858.119} C_VEL
LIN {X 0,Y 548.595,Z 1171.976,A -85,B 0,C 180,E1 25856.814,E2 25856.814} C_VEL
LIN {X 0,Y 547.719,Z 1190.947,A -85,B 0,C 180,E1 25855.363,E2 25855.363} C_VEL
LIN {X 0,Y 546.916,Z 1208.636,A -85,B 0,C 180,E1 25853.772,E2 25853.772} C_VEL
LIN {X 0,Y 546.225,Z 1224.249,A -85,B 0,C 180,E1 25852.147,E2 25852.147} C_VEL
LIN {X 0,Y 545.544,Z 1240.743,A -85,B 0,C 180,E1 25850.155,E2 25850.155} C_VEL
LIN {X 0,Y 545.004,Z 1254.987,A -85,B 0,C 180,E1 25848.138,E2 25848.138} C_VEL
LIN {X 0,Y 544.578,Z 1267.915,A -85,B 0,C 180,E1 25845.986,E2 25845.986} C_VEL
LIN {X 0,Y 544.304,Z 1278.36,A -85,B 0,C 180,E1 25843.925,E2 25843.925} C_VEL
LIN {X 0,Y 544.118,Z 1287.498,A -85,B 0,C 180,E1 25841.77,E2 25841.77} C_VEL
LIN {X 0,Y 544.002,Z 1295.223,A -85,B 0,C 180,E1 25839.522,E2 25839.522} C_VEL
LIN {X 0,Y 543.94,Z 1300.902,A -85,B 0,C 180,E1 25837.393,E2 25837.393} C_VEL
LIN {X 0,Y 543.91,Z 1305.485,A -85,B 0,C 180,E1 25835.063,E2 25835.063} C_VEL
LIN {X 0,Y 543.9,Z 1308.306,A -85,B 0,C 180,E1 25832.74,E2 25832.74} C_VEL
LIN {X 0,Y 543.895,Z 1309.373,A -85,B 0,C 180,E1 25830.632,E2 25830.632} C_VEL
LIN {X 0,Y 543.895,Z 1309.031,A -85,B 0,C 180,E1 25828.315,E2 25828.315} C_VEL
LIN {X 0,Y 543.899,Z 1307.121,A -85,B 0,C 180,E1 25826.1,E2 25826.1} C_VEL
LIN {X 0,Y 543.912,Z 1303.615,A -85,B 0,C 180,E1 25823.88,E2 25823.88} C_VEL
LIN {X 0,Y 543.956,Z 1298.592,A -85,B 0,C 180,E1 25821.651,E2 25821.651} C_VEL
LIN {X 0,Y 544.04,Z 1291.777,A -85,B 0,C 180,E1 25819.41,E2 25819.41} C_VEL
LIN {X 0,Y 544.195,Z 1283.165,A -85,B 0,C 180,E1 25817.156,E2 25817.156} C_VEL
LIN {X 0,Y 544.448,Z 1272.534,A -85,B 0,C 180,E1 25814.884,E2 25814.884} C_VEL
LIN {X 0,Y 544.777,Z 1261.611,A -85,B 0,C 180,E1 25812.924,E2 25812.924} C_VEL
LIN {X 0,Y 545.267,Z 1248.045,A -85,B 0,C 180,E1 25810.839,E2 25810.839} C_VEL
LIN {X 0,Y 545.865,Z 1232.798,A -85,B 0,C 180,E1 25808.849,E2 25808.849} C_VEL
LIN {X 0,Y 546.561,Z 1217.036,A -85,B 0,C 180,E1 25807.068,E2 25807.068} C_VEL
LIN {X 0,Y 547.39,Z 1198.384,A -85,B 0,C 180,E1 25805.274,E2 25805.274} C_VEL
LIN {X 0,Y 548.235,Z 1179.648,A -85,B 0,C 180,E1 25803.742,E2 25803.742} C_VEL
LIN {X 0,Y 549.12,Z 1160.142,A -85,B 0,C 180,E1 25802.394,E2 25802.394} C_VEL
LIN {X 0,Y 549.949,Z 1139.436,A -85,B 0,C 180,E1 25801.198,E2 25801.198} C_VEL
LIN {X 0,Y 550.765,Z 1118.159,A -85,B 0,C 180,E1 25800.199,E2 25800.199} C_VEL
LIN {X 0,Y 551.443,Z 1096.764,A -85,B 0,C 180,E1 25799.412,E2 25799.412} C_VEL
LIN {X 0,Y 551.985,Z 1074.787,A -85,B 0,C 180,E1 25798.806,E2 25798.806} C_VEL
LIN {X 0,Y 552.36,Z 1051.737,A -85,B 0,C 180,E1 25798.386,E2 25798.386} C_VEL
LIN {X 0,Y 554.166,Z 826.273,A -85,B 0,C 180,E1 25795.079,E2 25795.079} C_VEL
LIN {X 0,Y 554.621,Z 769.768,A -85,B 0,C 180,E1 25794.23,E2 25794.23} C_VEL
LIN {X 0,Y 555.939,Z 768.955,A -85,B 0,C 180,E1 25794.041,E2 25794.041} C_VEL
LIN {X 0,Y 557.779,Z 764.7,A -85,B 0,C 180,E1 25793.782,E2 25793.782} C_VEL
LIN {X 0,Y 559.129,Z 760.71,A -85,B 0,C 180,E1 25793.593,E2 25793.593} C_VEL
LIN {X 0,Y 563.068,Z 750.845,A -85,B 0,C 180,E1 25793.053,E2 25793.053} C_VEL
LIN {X 0,Y 566.239,Z 747.847,A -85,B 0,C 180,E1 25792.629,E2 25792.629} C_VEL
LIN {X 0,Y 567.06,Z 746.927,A -85,B 0,C 180,E1 25792.52,E2 25792.52} C_VEL
LIN {X 0,Y 568.218,Z 761.959,A -85,B 0,C 180,E1 25792.368,E2 25792.368} C_VEL
LIN {X 0,Y 570.399,Z 775.088,A -85,B 0,C 180,E1 25792.085,E2 25792.085} C_VEL
LIN {X 0,Y 573.601,Z 786.757,A -85,B 0,C 180,E1 25791.676,E2 25791.676} C_VEL
LIN {X 0,Y 577.732,Z 796.973,A -85,B 0,C 180,E1 25791.161,E2 25791.161} C_VEL
LIN {X 0,Y 582.782,Z 805.79,A -85,B 0,C 180,E1 25790.548,E2 25790.548} C_VEL
LIN {X 0,Y 586.536,Z 811.14,A -85,B 0,C 180,E1 25790.042,E2 25790.042} C_VEL
LIN {X 0,Y 588.361,Z 814.718,A -85,B 0,C 180,E1 25789.522,E2 25789.522} C_VEL
LIN {X 0,Y 588.761,Z 817.493,A -85,B 0,C 180,E1 25788.913,E2 25788.913} C_VEL
LIN {X 0,Y 587.722,Z 819.076,A -85,B 0,C 180,E1 25788.304,E2 25788.304} C_VEL
LIN {X 0,Y 585.35,Z 819.503,A -85,B 0,C 180,E1 25787.699,E2 25787.699} C_VEL
LIN {X 0,Y 582.107,Z 818.745,A -85,B 0,C 180,E1 25787.175,E2 25787.175} C_VEL
LIN {X 0,Y 576.283,Z 815.688,A -85,B 0,C 180,E1 25786.488,E2 25786.488} C_VEL
LIN {X 0,Y 569.649,Z 810.073,A -85,B 0,C 180,E1 25785.592,E2 25785.592} C_VEL
LIN {X 0,Y 564.454,Z 802.954,A -85,B 0,C 180,E1 25784.687,E2 25784.687} C_VEL
LIN {X 0,Y 560.679,Z 794.385,A -85,B 0,C 180,E1 25783.782,E2 25783.782} C_VEL
LIN {X 0,Y 558.206,Z 783.875,A -85,B 0,C 180,E1 25782.825,E2 25782.825} C_VEL
LIN {X 0,Y 557.099,Z 771.235,A -85,B 0,C 180,E1 25781.817,E2 25781.817} C_VEL
LIN {X 0,Y 557.799,Z 744.242,A -85,B 0,C 180,E1 25779.92,E2 25779.92} C_VEL
LIN {X 0,Y 559.411,Z 706.531,A -85,B 0,C 180,E1 25777.23,E2 25777.23} C_VEL
LIN {X 0,Y 559.784,Z 695.902,A -85,B 0,C 180,E1 25776.434,E2 25776.434} C_VEL
LIN {X 0,Y 552.006,Z 681.273,A -85,B 0,C 180,E1 25774.285,E2 25774.285} C_VEL
LIN {X 0,Y 548.723,Z 675.647,A -85,B 0,C 180,E1 25773.387,E2 25773.387} C_VEL
LIN {X 0,Y 546.713,Z 671.621,A -85,B 0,C 180,E1 25772.775,E2 25772.775} C_VEL
LIN {X 0,Y 544.845,Z 668.749,A -85,B 0,C 180,E1 25772.277,E2 25772.277} C_VEL
LIN {X 0,Y 544.404,Z 666.926,A -85,B 0,C 180,E1 25772.027,E2 25772.027} C_VEL
LIN {X 0,Y 544.41,Z 666.924,A -85,B 0,C 180,E1 25768.613,E2 25768.613} C_VEL
LIN {X 0,Y 544.392,Z 666.921,A -85,B 0,C 180,E1 25765.104,E2 25765.104} C_VEL
LIN {X 0,Y 544.395,Z 666.921,A -85,B 0,C 180,E1 25761.777,E2 25761.777} C_VEL
LIN {X 0,Y 544.39,Z 666.924,A -85,B 0,C 180,E1 25758.415,E2 25758.415} C_VEL
LIN {X 0,Y 544.403,Z 666.925,A -85,B 0,C 180,E1 25755.008,E2 25755.008} C_VEL
LIN {X 0,Y 544.403,Z 666.923,A -85,B 0,C 180,E1 25751.548,E2 25751.548} C_VEL
LIN {X 0,Y 544.4,Z 666.92,A -85,B 0,C 180,E1 25748.023,E2 25748.023} C_VEL
LIN {X 0,Y 544.402,Z 666.923,A -85,B 0,C 180,E1 25744.529,E2 25744.529} C_VEL
LIN {X 0,Y 544.404,Z 666.924,A -85,B 0,C 180,E1 25741.052,E2 25741.052} C_VEL
LIN {X 0,Y 544.387,Z 666.925,A -85,B 0,C 180,E1 25737.684,E2 25737.684} C_VEL
LIN {X 0,Y 544.396,Z 666.921,A -85,B 0,C 180,E1 25734.308,E2 25734.308} C_VEL
LIN {X 0,Y 544.401,Z 666.921,A -85,B 0,C 180,E1 25730.805,E2 25730.805} C_VEL
LIN {X 0,Y 544.407,Z 666.925,A -85,B 0,C 180,E1 25727.376,E2 25727.376} C_VEL
LIN {X 0,Y 544.399,Z 666.925,A -85,B 0,C 180,E1 25724.008,E2 25724.008} C_VEL
LIN {X 0,Y 544.386,Z 666.921,A -85,B 0,C 180,E1 25720.695,E2 25720.695} C_VEL
LIN {X 0,Y 544.384,Z 666.921,A -85,B 0,C 180,E1 25717.426,E2 25717.426} C_VEL
LIN {X 0,Y 544.385,Z 666.923,A -85,B 0,C 180,E1 25714.079,E2 25714.079} C_VEL
LIN {X 0,Y 544.386,Z 666.904,A -85,B 0,C 180,E1 25710.74,E2 25710.74} C_VEL
LIN {X 0,Y 544.397,Z 666.918,A -85,B 0,C 180,E1 25709.088,E2 25709.088} C_VEL
LIN {X 0,Y 543.391,Z 667.05,A -85,B 0,C 180,E1 25708.277,E2 25708.277} C_VEL
LIN {X 0,Y 536.983,Z 667.842,A -85,B 0,C 180,E1 25706,E2 25706} C_VEL
LIN {X 0,Y 536.45,Z 667.898,A -85,B 0,C 180,E1 25705.407,E2 25705.407} C_VEL
LIN {X 0,Y 536.458,Z 667.912,A -85,B 0,C 180,E1 25702.034,E2 25702.034} C_VEL
LIN {X 0,Y 536.462,Z 667.9,A -85,B 0,C 180,E1 25698.524,E2 25698.524} C_VEL
LIN {X 0,Y 536.467,Z 667.914,A -85,B 0,C 180,E1 25695.059,E2 25695.059} C_VEL
LIN {X 0,Y 536.462,Z 667.92,A -85,B 0,C 180,E1 25691.635,E2 25691.635} C_VEL
LIN {X 0,Y 536.478,Z 668.002,A -85,B 0,C 180,E1 25688.807,E2 25688.807} C_VEL
LIN {X 0,Y 537.661,Z 671.253,A -85,B 0,C 180,E1 25688.472,E2 25688.472} C_VEL
LIN {X 0,Y 545.311,Z 689.617,A -85,B 0,C 180,E1 25686.544,E2 25686.544} C_VEL
LIN {X 0,Y 544.072,Z 736.194,A -85,B 0,C 180,E1 25683.331,E2 25683.331} C_VEL
LIN {X 0,Y 543.178,Z 766.156,A -85,B 0,C 180,E1 25681.282,E2 25681.282} C_VEL
LIN {X 0,Y 544.935,Z 778.233,A -85,B 0,C 180,E1 25680.986,E2 25680.986} C_VEL
LIN {X 0,Y 543.109,Z 1013.78,A -85,B 0,C 180,E1 25677.599,E2 25677.599} C_VEL
LIN {X 0,Y 542.763,Z 1036.642,A -85,B 0,C 180,E1 25677.184,E2 25677.184} C_VEL
LIN {X 0,Y 542.246,Z 1057.352,A -85,B 0,C 180,E1 25676.603,E2 25676.603} C_VEL
LIN {X 0,Y 541.62,Z 1077.576,A -85,B 0,C 180,E1 25675.827,E2 25675.827} C_VEL
LIN {X 0,Y 540.912,Z 1096.612,A -85,B 0,C 180,E1 25674.894,E2 25674.894} C_VEL
LIN {X 0,Y 540.135,Z 1115.615,A -85,B 0,C 180,E1 25673.741,E2 25673.741} C_VEL
LIN {X 0,Y 539.331,Z 1133.908,A -85,B 0,C 180,E1 25672.393,E2 25672.393} C_VEL
LIN {X 0,Y 538.602,Z 1150.118,A -85,B 0,C 180,E1 25670.97,E2 25670.97} C_VEL
LIN {X 0,Y 537.928,Z 1165.34,A -85,B 0,C 180,E1 25669.402,E2 25669.402} C_VEL
LIN {X 0,Y 537.33,Z 1179.777,A -85,B 0,C 180,E1 25667.656,E2 25667.656} C_VEL
LIN {X 0,Y 536.847,Z 1192.923,A -85,B 0,C 180,E1 25665.778,E2 25665.778} C_VEL
LIN {X 0,Y 536.472,Z 1204.546,A -85,B 0,C 180,E1 25663.801,E2 25663.801} C_VEL
LIN {X 0,Y 536.21,Z 1214.659,A -85,B 0,C 180,E1 25661.727,E2 25661.727} C_VEL
LIN {X 0,Y 536.055,Z 1222.819,A -85,B 0,C 180,E1 25659.663,E2 25659.663} C_VEL
LIN {X 0,Y 535.962,Z 1229.485,A -85,B 0,C 180,E1 25657.503,E2 25657.503} C_VEL
LIN {X 0,Y 535.922,Z 1234.379,A -85,B 0,C 180,E1 25655.352,E2 25655.352} C_VEL
LIN {X 0,Y 535.913,Z 1237.733,A -85,B 0,C 180,E1 25653.101,E2 25653.101} C_VEL
LIN {X 0,Y 535.915,Z 1239.296,A -85,B 0,C 180,E1 25650.962,E2 25650.962} C_VEL
LIN {X 0,Y 535.909,Z 1239.27,A -85,B 0,C 180,E1 25648.824,E2 25648.824} C_VEL
LIN {X 0,Y 535.913,Z 1237.602,A -85,B 0,C 180,E1 25646.684,E2 25646.684} C_VEL
LIN {X 0,Y 535.925,Z 1234.344,A -85,B 0,C 180,E1 25644.54,E2 25644.54} C_VEL
LIN {X 0,Y 535.968,Z 1229.431,A -85,B 0,C 180,E1 25642.388,E2 25642.388} C_VEL
LIN {X 0,Y 536.056,Z 1222.745,A -85,B 0,C 180,E1 25640.227,E2 25640.227} C_VEL
LIN {X 0,Y 536.214,Z 1214.574,A -85,B 0,C 180,E1 25638.163,E2 25638.163} C_VEL
LIN {X 0,Y 536.459,Z 1204.919,A -85,B 0,C 180,E1 25636.18,E2 25636.18} C_VEL
LIN {X 0,Y 536.828,Z 1193.483,A -85,B 0,C 180,E1 25634.22,E2 25634.22} C_VEL
LIN {X 0,Y 537.311,Z 1180.264,A -85,B 0,C 180,E1 25632.319,E2 25632.319} C_VEL
LIN {X 0,Y 537.929,Z 1165.355,A -85,B 0,C 180,E1 25630.51,E2 25630.51} C_VEL
LIN {X 0,Y 538.621,Z 1149.597,A -85,B 0,C 180,E1 25628.892,E2 25628.892} C_VEL
LIN {X 0,Y 539.376,Z 1132.86,A -85,B 0,C 180,E1 25627.435,E2 25627.435} C_VEL
LIN {X 0,Y 540.163,Z 1114.903,A -85,B 0,C 180,E1 25626.123,E2 25626.123} C_VEL
LIN {X 0,Y 540.959,Z 1095.588,A -85,B 0,C 180,E1 25624.959,E2 25624.959} C_VEL
LIN {X 0,Y 541.678,Z 1076.127,A -85,B 0,C 180,E1 25624.018,E2 25624.018} C_VEL
LIN {X 0,Y 542.303,Z 1055.751,A -85,B 0,C 180,E1 25623.253,E2 25623.253} C_VEL
LIN {X 0,Y 542.783,Z 1035.109,A -85,B 0,C 180,E1 25622.69,E2 25622.69} C_VEL
LIN {X 0,Y 543.123,Z 1011.754,A -85,B 0,C 180,E1 25622.282,E2 25622.282} C_VEL
LIN {X 0,Y 544.905,Z 781.517,A -85,B 0,C 180,E1 25618.972,E2 25618.972} C_VEL
LIN {X 0,Y 541.749,Z 767.629,A -85,B 0,C 180,E1 25618.543,E2 25618.543} C_VEL
LIN {X 0,Y 542.82,Z 738.847,A -85,B 0,C 180,E1 25615.692,E2 25615.692} C_VEL
LIN {X 0,Y 543.781,Z 705.892,A -85,B 0,C 180,E1 25612.419,E2 25612.419} C_VEL
LIN {X 0,Y 544.204,Z 689.522,A -85,B 0,C 180,E1 25610.761,E2 25610.761} C_VEL
LIN {X 0,Y 538.721,Z 674.199,A -85,B 0,C 180,E1 25608.736,E2 25608.736} C_VEL
LIN {X 0,Y 536.459,Z 667.914,A -85,B 0,C 180,E1 25607.885,E2 25607.885} C_VEL
LIN {X 0,Y 536.46,Z 667.912,A -85,B 0,C 180,E1 25604.452,E2 25604.452} C_VEL
LIN {X 0,Y 536.448,Z 667.907,A -85,B 0,C 180,E1 25601.143,E2 25601.143} C_VEL
LIN {X 0,Y 536.457,Z 667.916,A -85,B 0,C 180,E1 25597.79,E2 25597.79} C_VEL
LIN {X 0,Y 536.474,Z 668.032,A -85,B 0,C 180,E1 25595.789,E2 25595.789} C_VEL
LIN {X 0,Y 544.223,Z 688.524,A -85,B 0,C 180,E1 25593.23,E2 25593.23} C_VEL
LIN {X 0,Y 542.655,Z 727.755,A -85,B 0,C 180,E1 25589.792,E2 25589.792} C_VEL
LIN {X 0,Y 541.114,Z 768.026,A -85,B 0,C 180,E1 25586.326,E2 25586.326} C_VEL
LIN {X 0,Y 539.628,Z 809.701,A -85,B 0,C 180,E1 25582.784,E2 25582.784} C_VEL
LIN {X 0,Y 538.842,Z 845.232,A -85,B 0,C 180,E1 25579.94,E2 25579.94} C_VEL
LIN {X 0,Y 539.995,Z 855.065,A -85,B 0,C 180,E1 25579.756,E2 25579.756} C_VEL
LIN {X 0,Y 539.147,Z 1014.068,A -85,B 0,C 180,E1 25577.557,E2 25577.557} C_VEL
LIN {X 0,Y 538.924,Z 1031.041,A -85,B 0,C 180,E1 25577.154,E2 25577.154} C_VEL
LIN {X 0,Y 538.578,Z 1047.466,A -85,B 0,C 180,E1 25576.557,E2 25576.557} C_VEL
LIN {X 0,Y 538.228,Z 1061.192,A -85,B 0,C 180,E1 25575.903,E2 25575.903} C_VEL
LIN {X 0,Y 537.864,Z 1074.137,A -85,B 0,C 180,E1 25575.14,E2 25575.14} C_VEL
LIN {X 0,Y 537.464,Z 1088.519,A -85,B 0,C 180,E1 25574.105,E2 25574.105} C_VEL
LIN {X 0,Y 537.022,Z 1102.947,A -85,B 0,C 180,E1 25572.801,E2 25572.801} C_VEL
LIN {X 0,Y 536.702,Z 1113.853,A -85,B 0,C 180,E1 25571.607,E2 25571.607} C_VEL
LIN {X 0,Y 536.425,Z 1124.638,A -85,B 0,C 180,E1 25570.2,E2 25570.2} C_VEL
LIN {X 0,Y 536.197,Z 1134.656,A -85,B 0,C 180,E1 25568.58,E2 25568.58} C_VEL
LIN {X 0,Y 536.059,Z 1142.156,A -85,B 0,C 180,E1 25567.071,E2 25567.071} C_VEL
LIN {X 0,Y 535.973,Z 1148.546,A -85,B 0,C 180,E1 25565.46,E2 25565.46} C_VEL
LIN {X 0,Y 535.93,Z 1154.21,A -85,B 0,C 180,E1 25563.509,E2 25563.509} C_VEL
LIN {X 0,Y 535.915,Z 1157.365,A -85,B 0,C 180,E1 25561.818,E2 25561.818} C_VEL
LIN {X 0,Y 535.915,Z 1159.11,A -85,B 0,C 180,E1 25560.107,E2 25560.107} C_VEL
LIN {X 0,Y 535.912,Z 1159.348,A -85,B 0,C 180,E1 25558.183,E2 25558.183} C_VEL
LIN {X 0,Y 535.916,Z 1157.744,A -85,B 0,C 180,E1 25556.363,E2 25556.363} C_VEL
LIN {X 0,Y 535.922,Z 1154.963,A -85,B 0,C 180,E1 25554.755,E2 25554.755} C_VEL
LIN {X 0,Y 535.963,Z 1150.281,A -85,B 0,C 180,E1 25552.964,E2 25552.964} C_VEL
LIN {X 0,Y 536.042,Z 1143.289,A -85,B 0,C 180,E1 25551.094,E2 25551.094} C_VEL
LIN {X 0,Y 536.168,Z 1135.973,A -85,B 0,C 180,E1 25549.579,E2 25549.579} C_VEL
LIN {X 0,Y 536.368,Z 1126.99,A -85,B 0,C 180,E1 25548.058,E2 25548.058} C_VEL
LIN {X 0,Y 536.653,Z 1115.796,A -85,B 0,C 180,E1 25546.533,E2 25546.533} C_VEL
LIN {X 0,Y 536.973,Z 1104.58,A -85,B 0,C 180,E1 25545.276,E2 25545.276} C_VEL
LIN {X 0,Y 537.345,Z 1092.322,A -85,B 0,C 180,E1 25544.126,E2 25544.126} C_VEL
LIN {X 0,Y 537.817,Z 1076.446,A -85,B 0,C 180,E1 25542.918,E2 25542.918} C_VEL
LIN {X 0,Y 538.185,Z 1062.801,A -85,B 0,C 180,E1 25542.093,E2 25542.093} C_VEL
LIN {X 0,Y 538.523,Z 1049.296,A -85,B 0,C 180,E1 25541.433,E2 25541.433} C_VEL
LIN {X 0,Y 538.886,Z 1033.108,A -85,B 0,C 180,E1 25540.821,E2 25540.821} C_VEL
LIN {X 0,Y 539.141,Z 1015.173,A -85,B 0,C 180,E1 25540.373,E2 25540.373} C_VEL
LIN {X 0,Y 539.446,Z 961.213,A -85,B 0,C 180,E1 25539.606,E2 25539.606} C_VEL
LIN {X 0,Y 539.795,Z 851.683,A -85,B 0,C 180,E1 25538.099,E2 25538.099} C_VEL
LIN {X 0,Y 538.808,Z 844.399,A -85,B 0,C 180,E1 25537.928,E2 25537.928} C_VEL
LIN {X 0,Y 539.637,Z 812.25,A -85,B 0,C 180,E1 25535.304,E2 25535.304} C_VEL
LIN {X 0,Y 542.348,Z 779.488,A -85,B 0,C 180,E1 25532.198,E2 25532.198} C_VEL
LIN {X 0,Y 546.146,Z 749.904,A -85,B 0,C 180,E1 25529.223,E2 25529.223} C_VEL
LIN {X 0,Y 550.515,Z 727.184,A -85,B 0,C 180,E1 25526.736,E2 25526.736} C_VEL
LIN {X 0,Y 554.956,Z 711.946,A -85,B 0,C 180,E1 25524.919,E2 25524.919} C_VEL
LIN {X 0,Y 557.898,Z 704.612,A -85,B 0,C 180,E1 25523.997,E2 25523.997} C_VEL
LIN {X 0,Y 557.759,Z 702.919,A -85,B 0,C 180,E1 25522.687,E2 25522.687} C_VEL
LIN {X 0,Y 551.62,Z 713.919,A -85,B 0,C 180,E1 25521.623,E2 25521.623} C_VEL
LIN {X 0,Y 547.401,Z 725.764,A -85,B 0,C 180,E1 25520.591,E2 25520.591} C_VEL
LIN {X 0,Y 544.641,Z 739.412,A -85,B 0,C 180,E1 25519.548,E2 25519.548} C_VEL
LIN {X 0,Y 543.372,Z 756.211,A -85,B 0,C 180,E1 25518.374,E2 25518.374} C_VEL
LIN {X 0,Y 544.183,Z 772.822,A -85,B 0,C 180,E1 25517.242,E2 25517.242} C_VEL
LIN {X 0,Y 546.855,Z 786.429,A -85,B 0,C 180,E1 25516.281,E2 25516.281} C_VEL
LIN {X 0,Y 551.199,Z 798.075,A -85,B 0,C 180,E1 25515.412,E2 25515.412} C_VEL
LIN {X 0,Y 556.706,Z 807.418,A -85,B 0,C 180,E1 25514.666,E2 25514.666} C_VEL
LIN {X 0,Y 563.803,Z 815.645,A -85,B 0,C 180,E1 25513.945,E2 25513.945} C_VEL
LIN {X 0,Y 572.515,Z 822.634,A -85,B 0,C 180,E1 25513.26,E2 25513.26} C_VEL
LIN {X 0,Y 577.001,Z 825.136,A -85,B 0,C 180,E1 25512.862,E2 25512.862} C_VEL
LIN {X 0,Y 580.794,Z 826.468,A -85,B 0,C 180,E1 25512.393,E2 25512.393} C_VEL
LIN {X 0,Y 583.84,Z 826.749,A -85,B 0,C 180,E1 25511.845,E2 25511.845} C_VEL
LIN {X 0,Y 585.679,Z 826.013,A -85,B 0,C 180,E1 25511.31,E2 25511.31} C_VEL
LIN {X 0,Y 586.47,Z 824.198,A -85,B 0,C 180,E1 25510.702,E2 25510.702} C_VEL
LIN {X 0,Y 585.823,Z 821.342,A -85,B 0,C 180,E1 25510.114,E2 25510.114} C_VEL
LIN {X 0,Y 583.666,Z 817.583,A -85,B 0,C 180,E1 25509.588,E2 25509.588} C_VEL
LIN {X 0,Y 577.894,Z 809.428,A -85,B 0,C 180,E1 25508.859,E2 25508.859} C_VEL
LIN {X 0,Y 572.756,Z 799.625,A -85,B 0,C 180,E1 25508.217,E2 25508.217} C_VEL
LIN {X 0,Y 568.643,Z 788.652,A -85,B 0,C 180,E1 25507.687,E2 25507.687} C_VEL
LIN {X 0,Y 565.524,Z 776.446,A -85,B 0,C 180,E1 25507.276,E2 25507.276} C_VEL
LIN {X 0,Y 563.525,Z 764.247,A -85,B 0,C 180,E1 25507.009,E2 25507.009} C_VEL
LIN {X 0,Y 561.836,Z 768.909,A -85,B 0,C 180,E1 25506.78,E2 25506.78} C_VEL
LIN {X 0,Y 559.488,Z 774.308,A -85,B 0,C 180,E1 25506.457,E2 25506.457} C_VEL
LIN {X 0,Y 558.923,Z 775.576,A -85,B 0,C 180,E1 25506.378,E2 25506.378} C_VEL
LIN {X 0,Y 554.736,Z 824.083,A -85,B 0,C 180,E1 25505.787,E2 25505.787} C_VEL
LIN {X 0,Y 550.961,Z 857.297,A -85,B 0,C 180,E1 25505.239,E2 25505.239} C_VEL
LIN {X 0,Y 548.591,Z 871.665,A -85,B 0,C 180,E1 25504.887,E2 25504.887} C_VEL
LIN {X 0,Y 547.414,Z 875.123,A -85,B 0,C 180,E1 25504.71,E2 25504.71} C_VEL
LIN {X 0,Y 547.131,Z 875.569,A -85,B 0,C 180,E1 25504.663,E2 25504.663} C_VEL
LIN {X 0,Y 545.35,Z 1065.522,A -85,B 0,C 180,E1 25501.826,E2 25501.826} C_VEL
LIN {X 0,Y 544.771,Z 1087.752,A -85,B 0,C 180,E1 25501.297,E2 25501.297} C_VEL
LIN {X 0,Y 544.053,Z 1110.309,A -85,B 0,C 180,E1 25500.541,E2 25500.541} C_VEL
LIN {X 0,Y 543.205,Z 1131.547,A -85,B 0,C 180,E1 25499.619,E2 25499.619} C_VEL
LIN {X 0,Y 542.289,Z 1151.777,A -85,B 0,C 180,E1 25498.525,E2 25498.525} C_VEL
LIN {X 0,Y 541.287,Z 1171.982,A -85,B 0,C 180,E1 25497.206,E2 25497.206} C_VEL
LIN {X 0,Y 540.254,Z 1191.719,A -85,B 0,C 180,E1 25495.671,E2 25495.671} C_VEL
LIN {X 0,Y 539.35,Z 1209.184,A -85,B 0,C 180,E1 25494.07,E2 25494.07} C_VEL
LIN {X 0,Y 538.552,Z 1224.972,A -85,B 0,C 180,E1 25492.397,E2 25492.397} C_VEL
LIN {X 0,Y 537.766,Z 1241.584,A -85,B 0,C 180,E1 25490.346,E2 25490.346} C_VEL
LIN {X 0,Y 537.158,Z 1255.553,A -85,B 0,C 180,E1 25488.323,E2 25488.323} C_VEL
LIN {X 0,Y 536.668,Z 1268.494,A -85,B 0,C 180,E1 25486.117,E2 25486.117} C_VEL
LIN {X 0,Y 536.374,Z 1278.356,A -85,B 0,C 180,E1 25484.135,E2 25484.135} C_VEL
LIN {X 0,Y 536.156,Z 1287.501,A -85,B 0,C 180,E1 25481.947,E2 25481.947} C_VEL
LIN {X 0,Y 536.012,Z 1295.529,A -85,B 0,C 180,E1 25479.557,E2 25479.557} C_VEL
LIN {X 0,Y 535.951,Z 1300.9,A -85,B 0,C 180,E1 25477.504,E2 25477.504} C_VEL
LIN {X 0,Y 535.913,Z 1305.488,A -85,B 0,C 180,E1 25475.138,E2 25475.138} C_VEL
LIN {X 0,Y 535.901,Z 1308.302,A -85,B 0,C 180,E1 25472.781,E2 25472.781} C_VEL
LIN {X 0,Y 535.895,Z 1309.373,A -85,B 0,C 180,E1 25470.642,E2 25470.642} C_VEL
LIN {X 0,Y 535.895,Z 1309.034,A -85,B 0,C 180,E1 25468.29,E2 25468.29} C_VEL
LIN {X 0,Y 535.9,Z 1307.117,A -85,B 0,C 180,E1 25466.042,E2 25466.042} C_VEL
LIN {X 0,Y 535.917,Z 1303.616,A -85,B 0,C 180,E1 25463.788,E2 25463.788} C_VEL
LIN {X 0,Y 535.969,Z 1298.592,A -85,B 0,C 180,E1 25461.526,E2 25461.526} C_VEL
LIN {X 0,Y 536.066,Z 1291.776,A -85,B 0,C 180,E1 25459.251,E2 25459.251} C_VEL
LIN {X 0,Y 536.25,Z 1283.169,A -85,B 0,C 180,E1 25456.962,E2 25456.962} C_VEL
LIN {X 0,Y 536.546,Z 1272.532,A -85,B 0,C 180,E1 25454.656,E2 25454.656} C_VEL
LIN {X 0,Y 536.918,Z 1261.607,A -85,B 0,C 180,E1 25452.666,E2 25452.666} C_VEL
LIN {X 0,Y 537.479,Z 1248.05,A -85,B 0,C 180,E1 25450.55,E2 25450.55} C_VEL
LIN {X 0,Y 538.157,Z 1233.051,A -85,B 0,C 180,E1 25448.563,E2 25448.563} C_VEL
LIN {X 0,Y 538.94,Z 1217.553,A -85,B 0,C 180,E1 25446.782,E2 25446.782} C_VEL
LIN {X 0,Y 539.89,Z 1199.007,A -85,B 0,C 180,E1 25444.965,E2 25444.965} C_VEL
LIN {X 0,Y 540.834,Z 1180.499,A -85,B 0,C 180,E1 25443.424,E2 25443.424} C_VEL
LIN {X 0,Y 541.843,Z 1161.04,A -85,B 0,C 180,E1 25442.05,E2 25442.05} C_VEL
LIN {X 0,Y 542.771,Z 1140.909,A -85,B 0,C 180,E1 25440.861,E2 25440.861} C_VEL
LIN {X 0,Y 543.676,Z 1120.242,A -85,B 0,C 180,E1 25439.864,E2 25439.864} C_VEL
LIN {X 0,Y 544.462,Z 1098.258,A -85,B 0,C 180,E1 25439.029,E2 25439.029} C_VEL
LIN {X 0,Y 545.094,Z 1076.511,A -85,B 0,C 180,E1 25438.409,E2 25438.409} C_VEL
LIN {X 0,Y 545.53,Z 1053.643,A -85,B 0,C 180,E1 25437.972,E2 25437.972} C_VEL
LIN {X 0,Y 547.267,Z 875.241,A -85,B 0,C 180,E1 25435.312,E2 25435.312} C_VEL
LIN {X 0,Y 548.265,Z 872.974,A -85,B 0,C 180,E1 25435.162,E2 25435.162} C_VEL
LIN {X 0,Y 550.362,Z 861.563,A -85,B 0,C 180,E1 25434.85,E2 25434.85} C_VEL
LIN {X 0,Y 553.983,Z 831.502,A -85,B 0,C 180,E1 25434.321,E2 25434.321} C_VEL
LIN {X 0,Y 558.186,Z 785.091,A -85,B 0,C 180,E1 25433.725,E2 25433.725} C_VEL
LIN {X 0,Y 559.112,Z 774.888,A -85,B 0,C 180,E1 25433.596,E2 25433.596} C_VEL
LIN {X 0,Y 561.495,Z 769.902,A -85,B 0,C 180,E1 25433.267,E2 25433.267} C_VEL
LIN {X 0,Y 563.369,Z 764.595,A -85,B 0,C 180,E1 25433.013,E2 25433.013} C_VEL
LIN {X 0,Y 563.576,Z 764.449,A -85,B 0,C 180,E1 25432.985,E2 25432.985} C_VEL
LIN {X 0,Y 565.86,Z 778.053,A -85,B 0,C 180,E1 25432.679,E2 25432.679} C_VEL
LIN {X 0,Y 569.173,Z 790.289,A -85,B 0,C 180,E1 25432.244,E2 25432.244} C_VEL
LIN {X 0,Y 573.446,Z 801.15,A -85,B 0,C 180,E1 25431.696,E2 25431.696} C_VEL
LIN {X 0,Y 578.673,Z 810.653,A -85,B 0,C 180,E1 25431.045,E2 25431.045} C_VEL
LIN {X 0,Y 583.79,Z 817.759,A -85,B 0,C 180,E1 25430.391,E2 25430.391} C_VEL
LIN {X 0,Y 585.867,Z 821.444,A -85,B 0,C 180,E1 25429.868,E2 25429.868} C_VEL
LIN {X 0,Y 586.463,Z 824.32,A -85,B 0,C 180,E1 25429.267,E2 25429.267} C_VEL
LIN {X 0,Y 585.542,Z 826.128,A -85,B 0,C 180,E1 25428.637,E2 25428.637} C_VEL
LIN {X 0,Y 583.371,Z 826.787,A -85,B 0,C 180,E1 25428.055,E2 25428.055} C_VEL
LIN {X 0,Y 579.816,Z 826.213,A -85,B 0,C 180,E1 25427.471,E2 25427.471} C_VEL
LIN {X 0,Y 574.301,Z 823.781,A -85,B 0,C 180,E1 25426.842,E2 25426.842} C_VEL
LIN {X 0,Y 567.345,Z 818.932,A -85,B 0,C 180,E1 25425.975,E2 25425.975} C_VEL
LIN {X 0,Y 561.187,Z 812.198,A -85,B 0,C 180,E1 25425.018,E2 25425.018} C_VEL
LIN {X 0,Y 556.476,Z 803.96,A -85,B 0,C 180,E1 25424.053,E2 25424.053} C_VEL
LIN {X 0,Y 553.059,Z 793.696,A -85,B 0,C 180,E1 25423.037,E2 25423.037} C_VEL
LIN {X 0,Y 551.139,Z 781.066,A -85,B 0,C 180,E1 25421.944,E2 25421.944} C_VEL
LIN {X 0,Y 550.86,Z 764.005,A -85,B 0,C 180,E1 25420.663,E2 25420.663} C_VEL
LIN {X 0,Y 552.918,Z 721.114,A -85,B 0,C 180,E1 25417.624,E2 25417.624} C_VEL
LIN {X 0,Y 553.776,Z 700.185,A -85,B 0,C 180,E1 25416.058,E2 25416.058} C_VEL
LIN {X 0,Y 545.739,Z 685.578,A -85,B 0,C 180,E1 25413.846,E2 25413.846} C_VEL
LIN {X 0,Y 543.258,Z 681.068,A -85,B 0,C 180,E1 25413.133,E2 25413.133} C_VEL
LIN {X 0,Y 541.184,Z 677.161,A -85,B 0,C 180,E1 25412.522,E2 25412.522} C_VEL
LIN {X 0,Y 539.171,Z 673.268,A -85,B 0,C 180,E1 25411.905,E2 25411.905} C_VEL
LIN {X 0,Y 536.854,Z 669.62,A -85,B 0,C 180,E1 25411.257,E2 25411.257} C_VEL
LIN {X 0,Y 536.451,Z 667.916,A -85,B 0,C 180,E1 25411.021,E2 25411.021} C_VEL
LIN {X 0,Y 536.463,Z 667.904,A -85,B 0,C 180,E1 25407.53,E2 25407.53} C_VEL
LIN {X 0,Y 536.458,Z 667.912,A -85,B 0,C 180,E1 25404.09,E2 25404.09} C_VEL
LIN {X 0,Y 536.451,Z 667.911,A -85,B 0,C 180,E1 25400.74,E2 25400.74} C_VEL
LIN {X 0,Y 536.448,Z 667.911,A -85,B 0,C 180,E1 25397.35,E2 25397.35} C_VEL
LIN {X 0,Y 536.448,Z 667.913,A -85,B 0,C 180,E1 25394.022,E2 25394.022} C_VEL
LIN {X 0,Y 536.459,Z 667.914,A -85,B 0,C 180,E1 25390.633,E2 25390.633} C_VEL
LIN {X 0,Y 536.47,Z 667.911,A -85,B 0,C 180,E1 25387.173,E2 25387.173} C_VEL
LIN {X 0,Y 536.457,Z 667.911,A -85,B 0,C 180,E1 25383.633,E2 25383.633} C_VEL
LIN {X 0,Y 536.454,Z 667.909,A -85,B 0,C 180,E1 25380.213,E2 25380.213} C_VEL
LIN {X 0,Y 536.451,Z 667.913,A -85,B 0,C 180,E1 25376.901,E2 25376.901} C_VEL
LIN {X 0,Y 536.463,Z 667.913,A -85,B 0,C 180,E1 25373.472,E2 25373.472} C_VEL
LIN {X 0,Y 536.465,Z 667.911,A -85,B 0,C 180,E1 25370.018,E2 25370.018} C_VEL
LIN {X 0,Y 536.461,Z 667.909,A -85,B 0,C 180,E1 25366.527,E2 25366.527} C_VEL
LIN {X 0,Y 536.463,Z 667.912,A -85,B 0,C 180,E1 25362.985,E2 25362.985} C_VEL
LIN {X 0,Y 536.466,Z 667.913,A -85,B 0,C 180,E1 25359.488,E2 25359.488} C_VEL
LIN {X 0,Y 536.45,Z 667.912,A -85,B 0,C 180,E1 25356.143,E2 25356.143} C_VEL
LIN {X 0,Y 536.46,Z 667.903,A -85,B 0,C 180,E1 25352.71,E2 25352.71} C_VEL
LIN {X 0,Y 536.461,Z 667.906,A -85,B 0,C 180,E1 25349.166,E2 25349.166} C_VEL
LIN {X 0,Y 536.465,Z 667.901,A -85,B 0,C 180,E1 25345.746,E2 25345.746} C_VEL
LIN {X 0,Y 536.45,Z 667.898,A -85,B 0,C 180,E1 25345.407,E2 25345.407} C_VEL
LIN {X 0,Y 535.459,Z 668.021,A -85,B 0,C 180,E1 25344.585,E2 25344.585} C_VEL
LIN {X 0,Y 529.054,Z 668.836,A -85,B 0,C 180,E1 25342.273,E2 25342.273} C_VEL
LIN {X 0,Y 528.526,Z 668.9,A -85,B 0,C 180,E1 25341.671,E2 25341.671} C_VEL
LIN {X 0,Y 528.519,Z 668.891,A -85,B 0,C 180,E1 25338.19,E2 25338.19} C_VEL
LIN {X 0,Y 528.516,Z 668.905,A -85,B 0,C 180,E1 25334.728,E2 25334.728} C_VEL
LIN {X 0,Y 528.521,Z 668.908,A -85,B 0,C 180,E1 25331.317,E2 25331.317} C_VEL
LIN {X 0,Y 528.529,Z 669.059,A -85,B 0,C 180,E1 25329.395,E2 25329.395} C_VEL
LIN {X 0,Y 529.557,Z 671.977,A -85,B 0,C 180,E1 25329.096,E2 25329.096} C_VEL
LIN {X 0,Y 536.822,Z 688.98,A -85,B 0,C 180,E1 25327.252,E2 25327.252} C_VEL
LIN {X 0,Y 538.438,Z 693.492,A -85,B 0,C 180,E1 25326.795,E2 25326.795} C_VEL
LIN {X 0,Y 536.959,Z 741.567,A -85,B 0,C 180,E1 25323.447,E2 25323.447} C_VEL
LIN {X 0,Y 536.239,Z 766.737,A -85,B 0,C 180,E1 25321.733,E2 25321.733} C_VEL
LIN {X 0,Y 538.096,Z 779.439,A -85,B 0,C 180,E1 25321.413,E2 25321.413} C_VEL
LIN {X 0,Y 536.021,Z 1014.213,A -85,B 0,C 180,E1 25317.99,E2 25317.99} C_VEL
LIN {X 0,Y 535.631,Z 1036.806,A -85,B 0,C 180,E1 25317.573,E2 25317.573} C_VEL
LIN {X 0,Y 535.05,Z 1057.767,A -85,B 0,C 180,E1 25316.975,E2 25316.975} C_VEL
LIN {X 0,Y 534.365,Z 1077.585,A -85,B 0,C 180,E1 25316.204,E2 25316.204} C_VEL
LIN {X 0,Y 533.546,Z 1097.134,A -85,B 0,C 180,E1 25315.231,E2 25315.231} C_VEL
LIN {X 0,Y 532.705,Z 1115.625,A -85,B 0,C 180,E1 25314.093,E2 25314.093} C_VEL
LIN {X 0,Y 531.799,Z 1133.965,A -85,B 0,C 180,E1 25312.724,E2 25312.724} C_VEL
LIN {X 0,Y 530.944,Z 1150.772,A -85,B 0,C 180,E1 25311.224,E2 25311.224} C_VEL
LIN {X 0,Y 530.178,Z 1166.07,A -85,B 0,C 180,E1 25309.614,E2 25309.614} C_VEL
LIN {X 0,Y 529.498,Z 1180.614,A -85,B 0,C 180,E1 25307.812,E2 25307.812} C_VEL
LIN {X 0,Y 528.956,Z 1193.622,A -85,B 0,C 180,E1 25305.907,E2 25305.907} C_VEL
LIN {X 0,Y 528.538,Z 1205.13,A -85,B 0,C 180,E1 25303.901,E2 25303.901} C_VEL
LIN {X 0,Y 528.243,Z 1215.125,A -85,B 0,C 180,E1 25301.795,E2 25301.795} C_VEL
LIN {X 0,Y 528.071,Z 1223.214,A -85,B 0,C 180,E1 25299.701,E2 25299.701} C_VEL
LIN {X 0,Y 527.967,Z 1229.787,A -85,B 0,C 180,E1 25297.508,E2 25297.508} C_VEL
LIN {X 0,Y 527.922,Z 1234.585,A -85,B 0,C 180,E1 25295.324,E2 25295.324} C_VEL
LIN {X 0,Y 527.912,Z 1237.846,A -85,B 0,C 180,E1 25293.039,E2 25293.039} C_VEL
LIN {X 0,Y 527.91,Z 1239.341,A -85,B 0,C 180,E1 25290.759,E2 25290.759} C_VEL
LIN {X 0,Y 527.901,Z 1239.168,A -85,B 0,C 180,E1 25288.589,E2 25288.589} C_VEL
LIN {X 0,Y 527.909,Z 1237.376,A -85,B 0,C 180,E1 25286.416,E2 25286.416} C_VEL
LIN {X 0,Y 527.932,Z 1233.932,A -85,B 0,C 180,E1 25284.239,E2 25284.239} C_VEL
LIN {X 0,Y 527.979,Z 1228.827,A -85,B 0,C 180,E1 25282.053,E2 25282.053} C_VEL
LIN {X 0,Y 528.087,Z 1221.939,A -85,B 0,C 180,E1 25279.858,E2 25279.858} C_VEL
LIN {X 0,Y 528.291,Z 1213.6,A -85,B 0,C 180,E1 25277.761,E2 25277.761} C_VEL
LIN {X 0,Y 528.608,Z 1203.276,A -85,B 0,C 180,E1 25275.653,E2 25275.653} C_VEL
LIN {X 0,Y 529.048,Z 1191.368,A -85,B 0,C 180,E1 25273.644,E2 25273.644} C_VEL
LIN {X 0,Y 529.629,Z 1177.866,A -85,B 0,C 180,E1 25271.73,E2 25271.73} C_VEL
LIN {X 0,Y 530.311,Z 1163.346,A -85,B 0,C 180,E1 25269.988,E2 25269.988} C_VEL
LIN {X 0,Y 531.107,Z 1147.192,A -85,B 0,C 180,E1 25268.346,E2 25268.346} C_VEL
LIN {X 0,Y 531.979,Z 1129.961,A -85,B 0,C 180,E1 25266.87,E2 25266.87} C_VEL
LIN {X 0,Y 532.876,Z 1111.674,A -85,B 0,C 180,E1 25265.56,E2 25265.56} C_VEL
LIN {X 0,Y 533.708,Z 1093.377,A -85,B 0,C 180,E1 25264.476,E2 25264.476} C_VEL
LIN {X 0,Y 534.496,Z 1074.367,A -85,B 0,C 180,E1 25263.562,E2 25263.562} C_VEL
LIN {X 0,Y 535.21,Z 1053.601,A -85,B 0,C 180,E1 25262.795,E2 25262.795} C_VEL
LIN {X 0,Y 535.732,Z 1032.588,A -85,B 0,C 180,E1 25262.239,E2 25262.239} C_VEL
LIN {X 0,Y 536.082,Z 1006.704,A -85,B 0,C 180,E1 25261.811,E2 25261.811} C_VEL
LIN {X 0,Y 538.054,Z 783.024,A -85,B 0,C 180,E1 25258.55,E2 25258.55} C_VEL
LIN {X 0,Y 534.648,Z 768.178,A -85,B 0,C 180,E1 25258.08,E2 25258.08} C_VEL
LIN {X 0,Y 535.796,Z 737.199,A -85,B 0,C 180,E1 25255.008,E2 25255.008} C_VEL
LIN {X 0,Y 536.896,Z 703.577,A -85,B 0,C 180,E1 25251.631,E2 25251.631} C_VEL
LIN {X 0,Y 537.137,Z 692.607,A -85,B 0,C 180,E1 25250.496,E2 25250.496} C_VEL
LIN {X 0,Y 531.374,Z 676.838,A -85,B 0,C 180,E1 25248.377,E2 25248.377} C_VEL
LIN {X 0,Y 528.511,Z 668.905,A -85,B 0,C 180,E1 25247.3,E2 25247.3} C_VEL
LIN {X 0,Y 528.527,Z 668.895,A -85,B 0,C 180,E1 25243.82,E2 25243.82} C_VEL
LIN {X 0,Y 528.529,Z 668.892,A -85,B 0,C 180,E1 25240.315,E2 25240.315} C_VEL
LIN {X 0,Y 528.512,Z 668.903,A -85,B 0,C 180,E1 25236.846,E2 25236.846} C_VEL
LIN {X 0,Y 528.529,Z 669.024,A -85,B 0,C 180,E1 25236.406,E2 25236.406} C_VEL
LIN {X 0,Y 537.238,Z 691.641,A -85,B 0,C 180,E1 25233.511,E2 25233.511} C_VEL
LIN {X 0,Y 535.617,Z 729.675,A -85,B 0,C 180,E1 25230.143,E2 25230.143} C_VEL
LIN {X 0,Y 533.935,Z 769.869,A -85,B 0,C 180,E1 25226.647,E2 25226.647} C_VEL
LIN {X 0,Y 532.428,Z 807.551,A -85,B 0,C 180,E1 25223.402,E2 25223.402} C_VEL
LIN {X 0,Y 531.178,Z 844.851,A -85,B 0,C 180,E1 25220.263,E2 25220.263} C_VEL
LIN {X 0,Y 532.513,Z 855.956,A -85,B 0,C 180,E1 25220.049,E2 25220.049} C_VEL
LIN {X 0,Y 531.562,Z 1013.956,A -85,B 0,C 180,E1 25217.833,E2 25217.833} C_VEL
LIN {X 0,Y 531.318,Z 1030.368,A -85,B 0,C 180,E1 25217.442,E2 25217.442} C_VEL
LIN {X 0,Y 530.914,Z 1047.811,A -85,B 0,C 180,E1 25216.803,E2 25216.803} C_VEL
LIN {X 0,Y 530.526,Z 1061.474,A -85,B 0,C 180,E1 25216.14,E2 25216.14} C_VEL
LIN {X 0,Y 530.121,Z 1074.372,A -85,B 0,C 180,E1 25215.367,E2 25215.367} C_VEL
LIN {X 0,Y 529.671,Z 1088.719,A -85,B 0,C 180,E1 25214.317,E2 25214.317} C_VEL
LIN {X 0,Y 529.189,Z 1102.562,A -85,B 0,C 180,E1 25213.049,E2 25213.049} C_VEL
LIN {X 0,Y 528.84,Z 1113.065,A -85,B 0,C 180,E1 25211.893,E2 25211.893} C_VEL
LIN {X 0,Y 528.534,Z 1123.185,A -85,B 0,C 180,E1 25210.574,E2 25210.574} C_VEL
LIN {X 0,Y 528.269,Z 1133.584,A -85,B 0,C 180,E1 25208.929,E2 25208.929} C_VEL
LIN {X 0,Y 528.088,Z 1141.742,A -85,B 0,C 180,E1 25207.288,E2 25207.288} C_VEL
LIN {X 0,Y 527.993,Z 1147.818,A -85,B 0,C 180,E1 25205.76,E2 25205.76} C_VEL
LIN {X 0,Y 527.94,Z 1153.138,A -85,B 0,C 180,E1 25204.018,E2 25204.018} C_VEL
LIN {X 0,Y 527.917,Z 1157.082,A -85,B 0,C 180,E1 25202.062,E2 25202.062} C_VEL
LIN {X 0,Y 527.914,Z 1158.966,A -85,B 0,C 180,E1 25200.326,E2 25200.326} C_VEL
LIN {X 0,Y 527.912,Z 1159.429,A -85,B 0,C 180,E1 25198.589,E2 25198.589} C_VEL
LIN {X 0,Y 527.915,Z 1158.016,A -85,B 0,C 180,E1 25196.526,E2 25196.526} C_VEL
LIN {X 0,Y 527.923,Z 1155.15,A -85,B 0,C 180,E1 25194.784,E2 25194.784} C_VEL
LIN {X 0,Y 527.959,Z 1151.056,A -85,B 0,C 180,E1 25193.148,E2 25193.148} C_VEL
LIN {X 0,Y 528.044,Z 1144.557,A -85,B 0,C 180,E1 25191.271,E2 25191.271} C_VEL
LIN {X 0,Y 528.182,Z 1137.031,A -85,B 0,C 180,E1 25189.64,E2 25189.64} C_VEL
LIN {X 0,Y 528.378,Z 1128.93,A -85,B 0,C 180,E1 25188.208,E2 25188.208} C_VEL
LIN {X 0,Y 528.689,Z 1118.316,A -85,B 0,C 180,E1 25186.66,E2 25186.66} C_VEL
LIN {X 0,Y 529.076,Z 1106.016,A -85,B 0,C 180,E1 25185.219,E2 25185.219} C_VEL
LIN {X 0,Y 529.455,Z 1094.615,A -85,B 0,C 180,E1 25184.108,E2 25184.108} C_VEL
LIN {X 0,Y 529.879,Z 1081.987,A -85,B 0,C 180,E1 25183.076,E2 25183.076} C_VEL
LIN {X 0,Y 530.393,Z 1066.562,A -85,B 0,C 180,E1 25182.048,E2 25182.048} C_VEL
LIN {X 0,Y 530.806,Z 1051.411,A -85,B 0,C 180,E1 25181.267,E2 25181.267} C_VEL
LIN {X 0,Y 531.15,Z 1037.565,A -85,B 0,C 180,E1 25180.709,E2 25180.709} C_VEL
LIN {X 0,Y 531.445,Z 1022.636,A -85,B 0,C 180,E1 25180.263,E2 25180.263} C_VEL
LIN {X 0,Y 531.686,Z 1002.994,A -85,B 0,C 180,E1 25179.898,E2 25179.898} C_VEL
LIN {X 0,Y 532.335,Z 852.747,A -85,B 0,C 180,E1 25177.808,E2 25177.808} C_VEL
LIN {X 0,Y 531.2,Z 844.594,A -85,B 0,C 180,E1 25177.624,E2 25177.624} C_VEL
LIN {X 0,Y 533.881,Z 807.171,A -85,B 0,C 180,E1 25174.128,E2 25174.128} C_VEL
LIN {X 0,Y 536.731,Z 779.08,A -85,B 0,C 180,E1 25171.396,E2 25171.396} C_VEL
LIN {X 0,Y 540.76,Z 752.469,A -85,B 0,C 180,E1 25168.641,E2 25168.641} C_VEL
LIN {X 0,Y 545.475,Z 731.436,A -85,B 0,C 180,E1 25166.262,E2 25166.262} C_VEL
LIN {X 0,Y 550.394,Z 716.826,A -85,B 0,C 180,E1 25164.457,E2 25164.457} C_VEL
LIN {X 0,Y 553.199,Z 710.695,A -85,B 0,C 180,E1 25163.642,E2 25163.642} C_VEL
LIN {X 0,Y 553.099,Z 710.044,A -85,B 0,C 180,E1 25163.037,E2 25163.037} C_VEL
LIN {X 0,Y 545.997,Z 721.731,A -85,B 0,C 180,E1 25161.871,E2 25161.871} C_VEL
LIN {X 0,Y 541.299,Z 733.563,A -85,B 0,C 180,E1 25160.794,E2 25160.794} C_VEL
LIN {X 0,Y 538.232,Z 747.062,A -85,B 0,C 180,E1 25159.7,E2 25159.7} C_VEL
LIN {X 0,Y 536.912,Z 762.463,A -85,B 0,C 180,E1 25158.546,E2 25158.546} C_VEL
LIN {X 0,Y 537.682,Z 778.085,A -85,B 0,C 180,E1 25157.4,E2 25157.4} C_VEL
LIN {X 0,Y 540.507,Z 791.745,A -85,B 0,C 180,E1 25156.371,E2 25156.371} C_VEL
LIN {X 0,Y 545.086,Z 803.487,A -85,B 0,C 180,E1 25155.443,E2 25155.443} C_VEL
LIN {X 0,Y 550.891,Z 812.996,A -85,B 0,C 180,E1 25154.645,E2 25154.645} C_VEL
LIN {X 0,Y 557.98,Z 821.124,A -85,B 0,C 180,E1 25153.917,E2 25153.917} C_VEL
LIN {X 0,Y 566.616,Z 828.174,A -85,B 0,C 180,E1 25153.21,E2 25153.21} C_VEL
LIN {X 0,Y 572.284,Z 831.591,A -85,B 0,C 180,E1 25152.795,E2 25152.795} C_VEL
LIN {X 0,Y 576.496,Z 833.323,A -85,B 0,C 180,E1 25152.367,E2 25152.367} C_VEL
LIN {X 0,Y 580.167,Z 834.029,A -85,B 0,C 180,E1 25151.833,E2 25151.833} C_VEL
LIN {X 0,Y 582.89,Z 833.499,A -85,B 0,C 180,E1 25151.201,E2 25151.201} C_VEL
LIN {X 0,Y 584.08,Z 831.882,A -85,B 0,C 180,E1 25150.58,E2 25150.58} C_VEL
LIN {X 0,Y 583.775,Z 829.173,A -85,B 0,C 180,E1 25149.962,E2 25149.962} C_VEL
LIN {X 0,Y 581.914,Z 825.637,A -85,B 0,C 180,E1 25149.412,E2 25149.412} C_VEL
LIN {X 0,Y 577.895,Z 820.317,A -85,B 0,C 180,E1 25148.859,E2 25148.859} C_VEL
LIN {X 0,Y 572.137,Z 811.222,A -85,B 0,C 180,E1 25148.138,E2 25148.138} C_VEL
LIN {X 0,Y 567.232,Z 800.637,A -85,B 0,C 180,E1 25147.503,E2 25147.503} C_VEL
LIN {X 0,Y 563.262,Z 788.649,A -85,B 0,C 180,E1 25146.973,E2 25146.973} C_VEL
LIN {X 0,Y 562.82,Z 787.311,A -85,B 0,C 180,E1 25146.913,E2 25146.913} C_VEL
LIN {X 0,Y 558.543,Z 833.563,A -85,B 0,C 180,E1 25146.325,E2 25146.325} C_VEL
LIN {X 0,Y 554.864,Z 863.519,A -85,B 0,C 180,E1 25145.805,E2 25145.805} C_VEL
LIN {X 0,Y 552.624,Z 875.656,A -85,B 0,C 180,E1 25145.482,E2 25145.482} C_VEL
LIN {X 0,Y 551.421,Z 879.974,A -85,B 0,C 180,E1 25145.306,E2 25145.306} C_VEL
LIN {X 0,Y 547.148,Z 931.763,A -85,B 0,C 180,E1 25144.669,E2 25144.669} C_VEL
LIN {X 0,Y 544.437,Z 951.706,A -85,B 0,C 180,E1 25144.352,E2 25144.352} C_VEL
LIN {X 0,Y 541.502,Z 965.535,A -85,B 0,C 180,E1 25144.004,E2 25144.004} C_VEL
LIN {X 0,Y 539.56,Z 972.967,A -85,B 0,C 180,E1 25143.68,E2 25143.68} C_VEL
LIN {X 0,Y 538.543,Z 1065.685,A -85,B 0,C 180,E1 25142.273,E2 25142.273} C_VEL
LIN {X 0,Y 537.913,Z 1087.622,A -85,B 0,C 180,E1 25141.746,E2 25141.746} C_VEL
LIN {X 0,Y 537.108,Z 1110.303,A -85,B 0,C 180,E1 25140.979,E2 25140.979} C_VEL
LIN {X 0,Y 536.16,Z 1131.419,A -85,B 0,C 180,E1 25140.054,E2 25140.054} C_VEL
LIN {X 0,Y 535.136,Z 1151.784,A -85,B 0,C 180,E1 25138.942,E2 25138.942} C_VEL
LIN {X 0,Y 534.006,Z 1171.987,A -85,B 0,C 180,E1 25137.608,E2 25137.608} C_VEL
LIN {X 0,Y 532.849,Z 1191.811,A -85,B 0,C 180,E1 25136.046,E2 25136.046} C_VEL
LIN {X 0,Y 531.833,Z 1209.176,A -85,B 0,C 180,E1 25134.432,E2 25134.432} C_VEL
LIN {X 0,Y 530.936,Z 1224.693,A -85,B 0,C 180,E1 25132.768,E2 25132.768} C_VEL
LIN {X 0,Y 530.072,Z 1240.75,A -85,B 0,C 180,E1 25130.77,E2 25130.77} C_VEL
LIN {X 0,Y 529.383,Z 1254.751,A -85,B 0,C 180,E1 25128.729,E2 25128.729} C_VEL
LIN {X 0,Y 528.839,Z 1267.526,A -85,B 0,C 180,E1 25126.552,E2 25126.552} C_VEL
LIN {X 0,Y 528.454,Z 1278.275,A -85,B 0,C 180,E1 25124.368,E2 25124.368} C_VEL
LIN {X 0,Y 528.198,Z 1287.505,A -85,B 0,C 180,E1 25122.13,E2 25122.13} C_VEL
LIN {X 0,Y 528.03,Z 1295.527,A -85,B 0,C 180,E1 25119.703,E2 25119.703} C_VEL
LIN {X 0,Y 527.962,Z 1300.898,A -85,B 0,C 180,E1 25117.618,E2 25117.618} C_VEL
LIN {X 0,Y 527.917,Z 1305.49,A -85,B 0,C 180,E1 25115.216,E2 25115.216} C_VEL
LIN {X 0,Y 527.901,Z 1308.298,A -85,B 0,C 180,E1 25112.823,E2 25112.823} C_VEL
LIN {X 0,Y 527.895,Z 1309.373,A -85,B 0,C 180,E1 25110.652,E2 25110.652} C_VEL
LIN {X 0,Y 527.896,Z 1309.036,A -85,B 0,C 180,E1 25108.264,E2 25108.264} C_VEL
LIN {X 0,Y 527.906,Z 1306.974,A -85,B 0,C 180,E1 25105.873,E2 25105.873} C_VEL
LIN {X 0,Y 527.923,Z 1303.618,A -85,B 0,C 180,E1 25103.694,E2 25103.694} C_VEL
LIN {X 0,Y 527.988,Z 1298.29,A -85,B 0,C 180,E1 25101.287,E2 25101.287} C_VEL
LIN {X 0,Y 528.105,Z 1291.398,A -85,B 0,C 180,E1 25098.976,E2 25098.976} C_VEL
LIN {X 0,Y 528.309,Z 1283.172,A -85,B 0,C 180,E1 25096.762,E2 25096.762} C_VEL
LIN {X 0,Y 528.649,Z 1272.529,A -85,B 0,C 180,E1 25094.421,E2 25094.421} C_VEL
LIN {X 0,Y 529.043,Z 1262.254,A -85,B 0,C 180,E1 25092.513,E2 25092.513} C_VEL
LIN {X 0,Y 529.67,Z 1248.83,A -85,B 0,C 180,E1 25090.367,E2 25090.367} C_VEL
LIN {X 0,Y 530.44,Z 1233.74,A -85,B 0,C 180,E1 25088.323,E2 25088.323} C_VEL
LIN {X 0,Y 531.266,Z 1219.085,A -85,B 0,C 180,E1 25086.603,E2 25086.603} C_VEL
LIN {X 0,Y 532.328,Z 1200.885,A -85,B 0,C 180,E1 25084.763,E2 25084.763} C_VEL
LIN {X 0,Y 533.415,Z 1181.956,A -85,B 0,C 180,E1 25083.145,E2 25083.145} C_VEL
LIN {X 0,Y 534.57,Z 1162.273,A -85,B 0,C 180,E1 25081.72,E2 25081.72} C_VEL
LIN {X 0,Y 535.593,Z 1142.749,A -85,B 0,C 180,E1 25080.535,E2 25080.535} C_VEL
LIN {X 0,Y 536.631,Z 1121.592,A -85,B 0,C 180,E1 25079.488,E2 25079.488} C_VEL
LIN {X 0,Y 537.511,Z 1099.638,A -85,B 0,C 180,E1 25078.633,E2 25078.633} C_VEL
LIN {X 0,Y 538.227,Z 1077.81,A -85,B 0,C 180,E1 25077.994,E2 25077.994} C_VEL
LIN {X 0,Y 538.716,Z 1055.432,A -85,B 0,C 180,E1 25077.549,E2 25077.549} C_VEL
LIN {X 0,Y 539.691,Z 971.981,A -85,B 0,C 180,E1 25076.286,E2 25076.286} C_VEL
LIN {X 0,Y 541.776,Z 964.412,A -85,B 0,C 180,E1 25075.959,E2 25075.959} C_VEL
LIN {X 0,Y 544.765,Z 949.847,A -85,B 0,C 180,E1 25075.613,E2 25075.613} C_VEL
LIN {X 0,Y 547.392,Z 929.14,A -85,B 0,C 180,E1 25075.294,E2 25075.294} C_VEL
LIN {X 0,Y 551.642,Z 878.815,A -85,B 0,C 180,E1 25074.661,E2 25074.661} C_VEL
LIN {X 0,Y 553.455,Z 871.9,A -85,B 0,C 180,E1 25074.398,E2 25074.398} C_VEL
LIN {X 0,Y 556.252,Z 853.342,A -85,B 0,C 180,E1 25073.997,E2 25073.997} C_VEL
LIN {X 0,Y 560.246,Z 816.629,A -85,B 0,C 180,E1 25073.439,E2 25073.439} C_VEL
LIN {X 0,Y 562.881,Z 787.252,A -85,B 0,C 180,E1 25073.079,E2 25073.079} C_VEL
LIN {X 0,Y 566.695,Z 799.241,A -85,B 0,C 180,E1 25072.568,E2 25072.568} C_VEL
LIN {X 0,Y 571.515,Z 810.042,A -85,B 0,C 180,E1 25071.942,E2 25071.942} C_VEL
LIN {X 0,Y 577.106,Z 819.215,A -85,B 0,C 180,E1 25071.238,E2 25071.238} C_VEL
LIN {X 0,Y 581.672,Z 825.277,A -85,B 0,C 180,E1 25070.634,E2 25070.634} C_VEL
LIN {X 0,Y 583.663,Z 828.87,A -85,B 0,C 180,E1 25070.094,E2 25070.094} C_VEL
LIN {X 0,Y 584.132,Z 831.558,A -85,B 0,C 180,E1 25069.511,E2 25069.511} C_VEL
LIN {X 0,Y 583.322,Z 833.191,A -85,B 0,C 180,E1 25068.955,E2 25068.955} C_VEL
LIN {X 0,Y 580.979,Z 834.033,A -85,B 0,C 180,E1 25068.323,E2 25068.323} C_VEL
LIN {X 0,Y 577.743,Z 833.667,A -85,B 0,C 180,E1 25067.792,E2 25067.792} C_VEL
LIN {X 0,Y 572.403,Z 831.691,A -85,B 0,C 180,E1 25067.192,E2 25067.192} C_VEL
LIN {X 0,Y 564.568,Z 826.968,A -85,B 0,C 180,E1 25066.267,E2 25066.267} C_VEL
LIN {X 0,Y 558.106,Z 820.964,A -85,B 0,C 180,E1 25065.335,E2 25065.335} C_VEL
LIN {X 0,Y 552.975,Z 813.782,A -85,B 0,C 180,E1 25064.407,E2 25064.407} C_VEL
LIN {X 0,Y 548.757,Z 804.49,A -85,B 0,C 180,E1 25063.386,E2 25063.386} C_VEL
LIN {X 0,Y 545.892,Z 793.033,A -85,B 0,C 180,E1 25062.3,E2 25062.3} C_VEL
LIN {X 0,Y 544.582,Z 779.478,A -85,B 0,C 180,E1 25061.171,E2 25061.171} C_VEL
LIN {X 0,Y 544.926,Z 761.047,A -85,B 0,C 180,E1 25059.819,E2 25059.819} C_VEL
LIN {X 0,Y 547.071,Z 721.367,A -85,B 0,C 180,E1 25056.963,E2 25056.963} C_VEL
LIN {X 0,Y 547.901,Z 704.95,A -85,B 0,C 180,E1 25055.73,E2 25055.73} C_VEL
LIN {X 0,Y 538.543,Z 687.647,A -85,B 0,C 180,E1 25053.082,E2 25053.082} C_VEL
LIN {X 0,Y 533.31,Z 678.214,A -85,B 0,C 180,E1 25051.538,E2 25051.538} C_VEL
LIN {X 0,Y 531.276,Z 674.429,A -85,B 0,C 180,E1 25050.916,E2 25050.916} C_VEL
LIN {X 0,Y 528.836,Z 670.378,A -85,B 0,C 180,E1 25050.193,E2 25050.193} C_VEL
LIN {X 0,Y 528.512,Z 668.905,A -85,B 0,C 180,E1 25049.963,E2 25049.963} C_VEL
LIN {X 0,Y 528.523,Z 668.895,A -85,B 0,C 180,E1 25046.516,E2 25046.516} C_VEL
LIN {X 0,Y 528.519,Z 668.901,A -85,B 0,C 180,E1 25042.936,E2 25042.936} C_VEL
LIN {X 0,Y 528.519,Z 668.903,A -85,B 0,C 180,E1 25039.563,E2 25039.563} C_VEL
LIN {X 0,Y 528.514,Z 668.901,A -85,B 0,C 180,E1 25036.147,E2 25036.147} C_VEL
LIN {X 0,Y 528.51,Z 668.901,A -85,B 0,C 180,E1 25032.788,E2 25032.788} C_VEL
LIN {X 0,Y 528.517,Z 668.901,A -85,B 0,C 180,E1 25029.363,E2 25029.363} C_VEL
LIN {X 0,Y 528.525,Z 668.901,A -85,B 0,C 180,E1 25025.863,E2 25025.863} C_VEL
LIN {X 0,Y 528.512,Z 668.902,A -85,B 0,C 180,E1 25022.385,E2 25022.385} C_VEL
LIN {X 0,Y 528.508,Z 668.901,A -85,B 0,C 180,E1 25019.024,E2 25019.024} C_VEL
LIN {X 0,Y 528.508,Z 668.9,A -85,B 0,C 180,E1 25015.66,E2 25015.66} C_VEL
LIN {X 0,Y 528.509,Z 668.903,A -85,B 0,C 180,E1 25012.28,E2 25012.28} C_VEL
LIN {X 0,Y 528.522,Z 668.901,A -85,B 0,C 180,E1 25008.874,E2 25008.874} C_VEL
LIN {X 0,Y 528.527,Z 668.901,A -85,B 0,C 180,E1 25005.427,E2 25005.427} C_VEL
LIN {X 0,Y 528.514,Z 668.899,A -85,B 0,C 180,E1 25001.925,E2 25001.925} C_VEL
LIN {X 0,Y 528.514,Z 668.902,A -85,B 0,C 180,E1 24998.468,E2 24998.468} C_VEL
LIN {X 0,Y 528.518,Z 668.903,A -85,B 0,C 180,E1 24995.047,E2 24995.047} C_VEL
LIN {X 0,Y 528.518,Z 668.878,A -85,B 0,C 180,E1 24991.604,E2 24991.604} C_VEL
LIN {X 0,Y 528.519,Z 668.9,A -85,B 0,C 180,E1 24988.014,E2 24988.014} C_VEL
LIN {X 0,Y 528.509,Z 668.882,A -85,B 0,C 180,E1 24984.624,E2 24984.624} C_VEL
LIN {X 0,Y 528.526,Z 668.9,A -85,B 0,C 180,E1 24981.671,E2 24981.671} C_VEL
LIN {X 0,Y 527.538,Z 669.022,A -85,B 0,C 180,E1 24980.836,E2 24980.836} C_VEL
LIN {X 0,Y 521.108,Z 669.811,A -85,B 0,C 180,E1 24978.491,E2 24978.491} C_VEL
LIN {X 0,Y 520.585,Z 669.882,A -85,B 0,C 180,E1 24977.879,E2 24977.879} C_VEL
LIN {X 0,Y 520.582,Z 669.893,A -85,B 0,C 180,E1 24974.355,E2 24974.355} C_VEL
LIN {X 0,Y 520.589,Z 669.897,A -85,B 0,C 180,E1 24970.768,E2 24970.768} C_VEL
LIN {X 0,Y 520.597,Z 669.99,A -85,B 0,C 180,E1 24970.003,E2 24970.003} C_VEL
LIN {X 0,Y 521.917,Z 673.431,A -85,B 0,C 180,E1 24969.634,E2 24969.634} C_VEL
LIN {X 0,Y 530,Z 692.471,A -85,B 0,C 180,E1 24967.541,E2 24967.541} C_VEL
LIN {X 0,Y 531.555,Z 697.067,A -85,B 0,C 180,E1 24967.074,E2 24967.074} C_VEL
LIN {X 0,Y 529.927,Z 745.322,A -85,B 0,C 180,E1 24963.687,E2 24963.687} C_VEL
LIN {X 0,Y 529.348,Z 767.435,A -85,B 0,C 180,E1 24962.192,E2 24962.192} C_VEL
LIN {X 0,Y 531.289,Z 780.699,A -85,B 0,C 180,E1 24961.85,E2 24961.85} C_VEL
LIN {X 0,Y 528.953,Z 1015.461,A -85,B 0,C 180,E1 24958.381,E2 24958.381} C_VEL
LIN {X 0,Y 528.516,Z 1037.427,A -85,B 0,C 180,E1 24957.961,E2 24957.961} C_VEL
LIN {X 0,Y 527.868,Z 1058.432,A -85,B 0,C 180,E1 24957.349,E2 24957.349} C_VEL
LIN {X 0,Y 527.134,Z 1077.594,A -85,B 0,C 180,E1 24956.592,E2 24956.592} C_VEL
LIN {X 0,Y 526.286,Z 1096.1,A -85,B 0,C 180,E1 24955.668,E2 24955.668} C_VEL
LIN {X 0,Y 525.338,Z 1114.755,A -85,B 0,C 180,E1 24954.513,E2 24954.513} C_VEL
LIN {X 0,Y 524.371,Z 1132.209,A -85,B 0,C 180,E1 24953.21,E2 24953.21} C_VEL
LIN {X 0,Y 523.43,Z 1148.673,A -85,B 0,C 180,E1 24951.751,E2 24951.751} C_VEL
LIN {X 0,Y 522.522,Z 1165.116,A -85,B 0,C 180,E1 24950.025,E2 24950.025} C_VEL
LIN {X 0,Y 521.753,Z 1179.782,A -85,B 0,C 180,E1 24948.201,E2 24948.201} C_VEL
LIN {X 0,Y 521.129,Z 1192.931,A -85,B 0,C 180,E1 24946.267,E2 24946.267} C_VEL
LIN {X 0,Y 520.651,Z 1204.558,A -85,B 0,C 180,E1 24944.229,E2 24944.229} C_VEL
LIN {X 0,Y 520.307,Z 1214.669,A -85,B 0,C 180,E1 24942.09,E2 24942.09} C_VEL
LIN {X 0,Y 520.093,Z 1223.216,A -85,B 0,C 180,E1 24939.851,E2 24939.851} C_VEL
LIN {X 0,Y 519.981,Z 1229.788,A -85,B 0,C 180,E1 24937.624,E2 24937.624} C_VEL
LIN {X 0,Y 519.927,Z 1234.586,A -85,B 0,C 180,E1 24935.407,E2 24935.407} C_VEL
LIN {X 0,Y 519.912,Z 1237.846,A -85,B 0,C 180,E1 24933.086,E2 24933.086} C_VEL
LIN {X 0,Y 519.91,Z 1239.341,A -85,B 0,C 180,E1 24930.771,E2 24930.771} C_VEL
LIN {X 0,Y 519.9,Z 1239.168,A -85,B 0,C 180,E1 24928.567,E2 24928.567} C_VEL
LIN {X 0,Y 519.91,Z 1237.375,A -85,B 0,C 180,E1 24926.361,E2 24926.361} C_VEL
LIN {X 0,Y 519.935,Z 1233.931,A -85,B 0,C 180,E1 24924.15,E2 24924.15} C_VEL
LIN {X 0,Y 519.986,Z 1228.825,A -85,B 0,C 180,E1 24921.93,E2 24921.93} C_VEL
LIN {X 0,Y 520.113,Z 1221.935,A -85,B 0,C 180,E1 24919.701,E2 24919.701} C_VEL
LIN {X 0,Y 520.349,Z 1213.595,A -85,B 0,C 180,E1 24917.572,E2 24917.572} C_VEL
LIN {X 0,Y 520.711,Z 1203.187,A -85,B 0,C 180,E1 24915.415,E2 24915.415} C_VEL
LIN {X 0,Y 521.206,Z 1191.366,A -85,B 0,C 180,E1 24913.391,E2 24913.391} C_VEL
LIN {X 0,Y 521.86,Z 1177.911,A -85,B 0,C 180,E1 24911.455,E2 24911.455} C_VEL
LIN {X 0,Y 522.628,Z 1163.336,A -85,B 0,C 180,E1 24909.681,E2 24909.681} C_VEL
LIN {X 0,Y 523.484,Z 1147.781,A -85,B 0,C 180,E1 24908.074,E2 24908.074} C_VEL
LIN {X 0,Y 524.448,Z 1130.672,A -85,B 0,C 180,E1 24906.577,E2 24906.577} C_VEL
LIN {X 0,Y 525.439,Z 1112.541,A -85,B 0,C 180,E1 24905.251,E2 24905.251} C_VEL
LIN {X 0,Y 526.377,Z 1094.117,A -85,B 0,C 180,E1 24904.136,E2 24904.136} C_VEL
LIN {X 0,Y 527.228,Z 1075.583,A -85,B 0,C 180,E1 24903.225,E2 24903.225} C_VEL
LIN {X 0,Y 527.994,Z 1055.375,A -85,B 0,C 180,E1 24902.456,E2 24902.456} C_VEL
LIN {X 0,Y 528.562,Z 1035.165,A -85,B 0,C 180,E1 24901.895,E2 24901.895} C_VEL
LIN {X 0,Y 528.988,Z 1011.752,A -85,B 0,C 180,E1 24901.475,E2 24901.475} C_VEL
LIN {X 0,Y 531.235,Z 784.61,A -85,B 0,C 180,E1 24898.118,E2 24898.118} C_VEL
LIN {X 0,Y 527.551,Z 768.613,A -85,B 0,C 180,E1 24897.602,E2 24897.602} C_VEL
LIN {X 0,Y 528.654,Z 739.442,A -85,B 0,C 180,E1 24894.704,E2 24894.704} C_VEL
LIN {X 0,Y 529.894,Z 705.721,A -85,B 0,C 180,E1 24891.28,E2 24891.28} C_VEL
LIN {X 0,Y 530.122,Z 695.908,A -85,B 0,C 180,E1 24890.254,E2 24890.254} C_VEL
LIN {X 0,Y 524.288,Z 679.741,A -85,B 0,C 180,E1 24888.053,E2 24888.053} C_VEL
LIN {X 0,Y 520.582,Z 669.891,A -85,B 0,C 180,E1 24886.673,E2 24886.673} C_VEL
LIN {X 0,Y 520.572,Z 669.883,A -85,B 0,C 180,E1 24883.285,E2 24883.285} C_VEL
LIN {X 0,Y 520.583,Z 669.884,A -85,B 0,C 180,E1 24879.904,E2 24879.904} C_VEL
LIN {X 0,Y 520.59,Z 669.954,A -85,B 0,C 180,E1 24877.053,E2 24877.053} C_VEL
LIN {X 0,Y 529.38,Z 692.546,A -85,B 0,C 180,E1 24874.084,E2 24874.084} C_VEL
LIN {X 0,Y 530.311,Z 695.257,A -85,B 0,C 180,E1 24873.75,E2 24873.75} C_VEL
LIN {X 0,Y 528.522,Z 733.515,A -85,B 0,C 180,E1 24870.339,E2 24870.339} C_VEL
LIN {X 0,Y 526.722,Z 773.242,A -85,B 0,C 180,E1 24866.85,E2 24866.85} C_VEL
LIN {X 0,Y 525.023,Z 813.242,A -85,B 0,C 180,E1 24863.375,E2 24863.375} C_VEL
LIN {X 0,Y 523.839,Z 846.181,A -85,B 0,C 180,E1 24860.582,E2 24860.582} C_VEL
LIN {X 0,Y 525.09,Z 856.818,A -85,B 0,C 180,E1 24860.364,E2 24860.364} C_VEL
LIN {X 0,Y 523.992,Z 1013.844,A -85,B 0,C 180,E1 24858.118,E2 24858.118} C_VEL
LIN {X 0,Y 523.726,Z 1029.393,A -85,B 0,C 180,E1 24857.747,E2 24857.747} C_VEL
LIN {X 0,Y 523.3,Z 1046.917,A -85,B 0,C 180,E1 24857.112,E2 24857.112} C_VEL
LIN {X 0,Y 522.868,Z 1060.743,A -85,B 0,C 180,E1 24856.44,E2 24856.44} C_VEL
LIN {X 0,Y 522.415,Z 1073.757,A -85,B 0,C 180,E1 24855.656,E2 24855.656} C_VEL
LIN {X 0,Y 521.95,Z 1086.769,A -85,B 0,C 180,E1 24854.704,E2 24854.704} C_VEL
LIN {X 0,Y 521.393,Z 1101.624,A -85,B 0,C 180,E1 24853.363,E2 24853.363} C_VEL
LIN {X 0,Y 520.992,Z 1112.277,A -85,B 0,C 180,E1 24852.187,E2 24852.187} C_VEL
LIN {X 0,Y 520.667,Z 1121.718,A -85,B 0,C 180,E1 24850.96,E2 24850.96} C_VEL
LIN {X 0,Y 520.398,Z 1130.407,A -85,B 0,C 180,E1 24849.623,E2 24849.623} C_VEL
LIN {X 0,Y 520.171,Z 1139.359,A -85,B 0,C 180,E1 24847.955,E2 24847.955} C_VEL
LIN {X 0,Y 520.025,Z 1146.702,A -85,B 0,C 180,E1 24846.181,E2 24846.181} C_VEL
LIN {X 0,Y 519.955,Z 1151.656,A -85,B 0,C 180,E1 24844.633,E2 24844.633} C_VEL
LIN {X 0,Y 519.922,Z 1155.58,A -85,B 0,C 180,E1 24842.977,E2 24842.977} C_VEL
LIN {X 0,Y 519.913,Z 1158.511,A -85,B 0,C 180,E1 24840.992,E2 24840.992} C_VEL
LIN {X 0,Y 519.915,Z 1159.422,A -85,B 0,C 180,E1 24839.119,E2 24839.119} C_VEL
LIN {X 0,Y 519.916,Z 1158.894,A -85,B 0,C 180,E1 24837.465,E2 24837.465} C_VEL
LIN {X 0,Y 519.917,Z 1156.939,A -85,B 0,C 180,E1 24835.699,E2 24835.699} C_VEL
LIN {X 0,Y 519.944,Z 1152.846,A -85,B 0,C 180,E1 24833.707,E2 24833.707} C_VEL
LIN {X 0,Y 520.006,Z 1147.805,A -85,B 0,C 180,E1 24832.043,E2 24832.043} C_VEL
LIN {X 0,Y 520.119,Z 1141.696,A -85,B 0,C 180,E1 24830.484,E2 24830.484} C_VEL
LIN {X 0,Y 520.321,Z 1133.485,A -85,B 0,C 180,E1 24828.809,E2 24828.809} C_VEL
LIN {X 0,Y 520.601,Z 1123.766,A -85,B 0,C 180,E1 24827.24,E2 24827.24} C_VEL
LIN {X 0,Y 520.938,Z 1113.665,A -85,B 0,C 180,E1 24825.892,E2 24825.892} C_VEL
LIN {X 0,Y 521.316,Z 1103.442,A -85,B 0,C 180,E1 24824.738,E2 24824.738} C_VEL
LIN {X 0,Y 521.832,Z 1090.312,A -85,B 0,C 180,E1 24823.492,E2 24823.492} C_VEL
LIN {X 0,Y 522.35,Z 1075.912,A -85,B 0,C 180,E1 24822.396,E2 24822.396} C_VEL
LIN {X 0,Y 522.783,Z 1063.193,A -85,B 0,C 180,E1 24821.605,E2 24821.605} C_VEL
LIN {X 0,Y 523.206,Z 1049.777,A -85,B 0,C 180,E1 24820.927,E2 24820.927} C_VEL
